LIN {X 0,Y 520.9,Z 965.477,A -85,B 0,C 180,E1 12388.23,E2 12388.23} C_VEL
LIN {X 0,Y 527.511,Z 989.341,A -85,B 0,C 180,E1 12389.551,E2 12389.551} C_VEL
LIN {X 0,Y 523.84,Z 1027.553,A -85,B 0,C 180,E1 12391.504,E2 12391.504} C_VEL
LIN {X 0,Y 519.786,Z 1062.879,A -85,B 0,C 180,E1 12394.029,E2 12394.029} C_VEL
LIN {X 0,Y 515.868,Z 1094.861,A -85,B 0,C 180,E1 12397.118,E2 12397.118} C_VEL
LIN {X 0,Y 512.363,Z 1122.894,A -85,B 0,C 180,E1 12400.744,E2 12400.744} C_VEL
LIN {X 0,Y 509.855,Z 1145.557,A -85,B 0,C 180,E1 12404.748,E2 12404.748} C_VEL
LIN {X 0,Y 508.379,Z 1161.603,A -85,B 0,C 180,E1 12408.676,E2 12408.676} C_VEL
LIN {X 0,Y 507.524,Z 1173.609,A -85,B 0,C 180,E1 12413.158,E2 12413.158} C_VEL
LIN {X 0,Y 507.269,Z 1178.777,A -85,B 0,C 180,E1 12416.583,E2 12416.583} C_VEL
LIN {X 0,Y 507.149,Z 1180.724,A -85,B 0,C 180,E1 12419.998,E2 12419.998} C_VEL
LIN {X 0,Y 507.304,Z 1179.309,A -85,B 0,C 180,E1 12423.414,E2 12423.414} C_VEL
LIN {X 0,Y 507.847,Z 1172.983,A -85,B 0,C 180,E1 12427.693,E2 12427.693} C_VEL
LIN {X 0,Y 508.836,Z 1161.151,A -85,B 0,C 180,E1 12431.996,E2 12431.996} C_VEL
LIN {X 0,Y 510.794,Z 1143.685,A -85,B 0,C 180,E1 12436.18,E2 12436.18} C_VEL
LIN {X 0,Y 513.724,Z 1121.065,A -85,B 0,C 180,E1 12440.059,E2 12440.059} C_VEL
LIN {X 0,Y 517.458,Z 1094.082,A -85,B 0,C 180,E1 12443.494,E2 12443.494} C_VEL
LIN {X 0,Y 521.913,Z 1061.989,A -85,B 0,C 180,E1 12446.546,E2 12446.546} C_VEL
LIN {X 0,Y 526.403,Z 1024.953,A -85,B 0,C 180,E1 12449.129,E2 12449.129} C_VEL
LIN {X 0,Y 529.643,Z 987.235,A -85,B 0,C 180,E1 12451.052,E2 12451.052} C_VEL
LIN {X 0,Y 522.519,Z 958.525,A -85,B 0,C 180,E1 12452.917,E2 12452.917} C_VEL
LIN {X 0,Y 511.608,Z 934.411,A -85,B 0,C 180,E1 12454.931,E2 12454.931} C_VEL
LIN {X 0,Y 505.831,Z 924.14,A -85,B 0,C 180,E1 12456.044,E2 12456.044} C_VEL
LIN {X 0,Y 505.742,Z 923.03,A -85,B 0,C 180,E1 12456.255,E2 12456.255} C_VEL
LIN {X 0,Y 505.562,Z 923.03,A -85,B 0,C 180,E1 12461.677,E2 12461.677} C_VEL
LIN {X 0,Y 505.58,Z 923.03,A -85,B 0,C 180,E1 12468.346,E2 12468.346} C_VEL
LIN {X 0,Y 505.778,Z 923.5,A -85,B 0,C 180,E1 12473,E2 12473} C_VEL
LIN {X 0,Y 508.487,Z 928.998,A -85,B 0,C 180,E1 12473.585,E2 12473.585} C_VEL
LIN {X 0,Y 520.191,Z 951.391,A -85,B 0,C 180,E1 12475.641,E2 12475.641} C_VEL
LIN {X 0,Y 529.457,Z 976.982,A -85,B 0,C 180,E1 12477.182,E2 12477.182} C_VEL
LIN {X 0,Y 531.635,Z 989.961,A -85,B 0,C 180,E1 12477.756,E2 12477.756} C_VEL
LIN {X 0,Y 527.643,Z 1032.457,A -85,B 0,C 180,E1 12479.219,E2 12479.219} C_VEL
LIN {X 0,Y 523.137,Z 1072.758,A -85,B 0,C 180,E1 12481.282,E2 12481.282} C_VEL
LIN {X 0,Y 518.67,Z 1110.607,A -85,B 0,C 180,E1 12483.99,E2 12483.99} C_VEL
LIN {X 0,Y 514.873,Z 1141.401,A -85,B 0,C 180,E1 12486.934,E2 12486.934} C_VEL
LIN {X 0,Y 509.62,Z 1153.637,A -85,B 0,C 180,E1 12488.212,E2 12488.212} C_VEL
LIN {X 0,Y 504.32,Z 1165.107,A -85,B 0,C 180,E1 12489.59,E2 12489.59} C_VEL
LIN {X 0,Y 501.753,Z 1188.474,A -85,B 0,C 180,E1 12493.393,E2 12493.393} C_VEL
LIN {X 0,Y 500.297,Z 1206.459,A -85,B 0,C 180,E1 12497.368,E2 12497.368} C_VEL
LIN {X 0,Y 499.642,Z 1218.968,A -85,B 0,C 180,E1 12501.319,E2 12501.319} C_VEL
LIN {X 0,Y 499.431,Z 1227.195,A -85,B 0,C 180,E1 12505.678,E2 12505.678} C_VEL
LIN {X 0,Y 499.394,Z 1229.924,A -85,B 0,C 180,E1 12510.015,E2 12510.015} C_VEL
LIN {X 0,Y 499.406,Z 1227.246,A -85,B 0,C 180,E1 12514.353,E2 12514.353} C_VEL
LIN {X 0,Y 499.659,Z 1219.037,A -85,B 0,C 180,E1 12518.712,E2 12518.712} C_VEL
LIN {X 0,Y 500.448,Z 1204.807,A -85,B 0,C 180,E1 12523.103,E2 12523.103} C_VEL
LIN {X 0,Y 502.2,Z 1184.844,A -85,B 0,C 180,E1 12527.3,E2 12527.3} C_VEL
LIN {X 0,Y 504.951,Z 1160.393,A -85,B 0,C 180,E1 12531.059,E2 12531.059} C_VEL
LIN {X 0,Y 508.606,Z 1130.776,A -85,B 0,C 180,E1 12534.476,E2 12534.476} C_VEL
LIN {X 0,Y 512.785,Z 1097.991,A -85,B 0,C 180,E1 12537.311,E2 12537.311} C_VEL
LIN {X 0,Y 517.104,Z 1059.799,A -85,B 0,C 180,E1 12539.735,E2 12539.735} C_VEL
LIN {X 0,Y 520.912,Z 1019.258,A -85,B 0,C 180,E1 12541.491,E2 12541.491} C_VEL
LIN {X 0,Y 522.653,Z 988.371,A -85,B 0,C 180,E1 12542.388,E2 12542.388} C_VEL
LIN {X 0,Y 497.906,Z 923.03,A -85,B 0,C 180,E1 12545.137,E2 12545.137} C_VEL
LIN {X 0,Y 497.67,Z 923.03,A -85,B 0,C 180,E1 12551.928,E2 12551.928} C_VEL
LIN {X 0,Y 497.676,Z 923.03,A -85,B 0,C 180,E1 12558.091,E2 12558.091} C_VEL
LIN {X 0,Y 497.784,Z 923.03,A -85,B 0,C 180,E1 12564.778,E2 12564.778} C_VEL
LIN {X 0,Y 497.927,Z 923.03,A -85,B 0,C 180,E1 12570.953,E2 12570.953} C_VEL
LIN {X 0,Y 498.06,Z 923.03,A -85,B 0,C 180,E1 12576.773,E2 12576.773} C_VEL
LIN {X 0,Y 498.161,Z 923.03,A -85,B 0,C 180,E1 12582.344,E2 12582.344} C_VEL
LIN {X 0,Y 498.445,Z 923.03,A -85,B 0,C 180,E1 12587.75,E2 12587.75} C_VEL
LIN {X 0,Y 498.675,Z 923.03,A -85,B 0,C 180,E1 12590.677,E2 12590.677} C_VEL
LIN {X 0,Y 508.907,Z 958.608,A -85,B 0,C 180,E1 12591.929,E2 12591.929} C_VEL
LIN {X 0,Y 508.728,Z 999.028,A -85,B 0,C 180,E1 12592.833,E2 12592.833} C_VEL
LIN {X 0,Y 507.812,Z 1027.625,A -85,B 0,C 180,E1 12594.131,E2 12594.131} C_VEL
LIN {X 0,Y 506.287,Z 1053.415,A -85,B 0,C 180,E1 12596.044,E2 12596.044} C_VEL
LIN {X 0,Y 504.623,Z 1075.233,A -85,B 0,C 180,E1 12598.5,E2 12598.5} C_VEL
LIN {X 0,Y 503.071,Z 1091.622,A -85,B 0,C 180,E1 12601.293,E2 12601.293} C_VEL
LIN {X 0,Y 501.81,Z 1102.595,A -85,B 0,C 180,E1 12604.319,E2 12604.319} C_VEL
LIN {X 0,Y 501.149,Z 1107.533,A -85,B 0,C 180,E1 12606.929,E2 12606.929} C_VEL
LIN {X 0,Y 500.871,Z 1108.785,A -85,B 0,C 180,E1 12608.678,E2 12608.678} C_VEL
LIN {X 0,Y 500.809,Z 1107.29,A -85,B 0,C 180,E1 12611.485,E2 12611.485} C_VEL
LIN {X 0,Y 501.096,Z 1100.753,A -85,B 0,C 180,E1 12614.58,E2 12614.58} C_VEL
LIN {X 0,Y 501.602,Z 1089.12,A -85,B 0,C 180,E1 12617.535,E2 12617.535} C_VEL
LIN {X 0,Y 502.57,Z 1070.875,A -85,B 0,C 180,E1 12620.461,E2 12620.461} C_VEL
LIN {X 0,Y 503.728,Z 1048.712,A -85,B 0,C 180,E1 12622.843,E2 12622.843} C_VEL
LIN {X 0,Y 504.947,Z 1021.724,A -85,B 0,C 180,E1 12624.771,E2 12624.771} C_VEL
LIN {X 0,Y 505.662,Z 992.567,A -85,B 0,C 180,E1 12626.047,E2 12626.047} C_VEL
LIN {X 0,Y 505.274,Z 955.718,A -85,B 0,C 180,E1 12626.834,E2 12626.834} C_VEL
LIN {X 0,Y 498.179,Z 923.03,A -85,B 0,C 180,E1 12627.573,E2 12627.573} C_VEL
LIN {X 0,Y 497.791,Z 923.03,A -85,B 0,C 180,E1 12633.123,E2 12633.123} C_VEL
LIN {X 0,Y 497.681,Z 923.03,A -85,B 0,C 180,E1 12639.617,E2 12639.617} C_VEL
LIN {X 0,Y 497.669,Z 923.03,A -85,B 0,C 180,E1 12645.688,E2 12645.688} C_VEL
LIN {X 0,Y 497.713,Z 923.03,A -85,B 0,C 180,E1 12652.131,E2 12652.131} C_VEL
LIN {X 0,Y 497.801,Z 923.03,A -85,B 0,C 180,E1 12658.21,E2 12658.21} C_VEL
LIN {X 0,Y 498.065,Z 923.03,A -85,B 0,C 180,E1 12662.915,E2 12662.915} C_VEL
LIN {X 0,Y 498.194,Z 923.03,A -85,B 0,C 180,E1 12668.641,E2 12668.641} C_VEL
LIN {X 0,Y 498.358,Z 923.03,A -85,B 0,C 180,E1 12674.149,E2 12674.149} C_VEL
LIN {X 0,Y 498.609,Z 923.03,A -85,B 0,C 180,E1 12679.509,E2 12679.509} C_VEL
LIN {X 0,Y 498.918,Z 923.03,A -85,B 0,C 180,E1 12684.772,E2 12684.772} C_VEL
LIN {X 0,Y 499.243,Z 923.03,A -85,B 0,C 180,E1 12689.985,E2 12689.985} C_VEL
LIN {X 0,Y 498.995,Z 923.03,A -85,B 0,C 180,E1 12695.197,E2 12695.197} C_VEL
LIN {X 0,Y 498.647,Z 923.03,A -85,B 0,C 180,E1 12700.459,E2 12700.459} C_VEL
LIN {X 0,Y 498.446,Z 923.03,A -85,B 0,C 180,E1 12705.816,E2 12705.816} C_VEL
LIN {X 0,Y 498.223,Z 923.03,A -85,B 0,C 180,E1 12711.325,E2 12711.325} C_VEL
LIN {X 0,Y 498.034,Z 923.03,A -85,B 0,C 180,E1 12717.053,E2 12717.053} C_VEL
LIN {X 0,Y 497.906,Z 923.03,A -85,B 0,C 180,E1 12723.091,E2 12723.091} C_VEL
LIN {X 0,Y 497.714,Z 923.03,A -85,B 0,C 180,E1 12729.587,E2 12729.587} C_VEL
LIN {X 0,Y 497.783,Z 923.03,A -85,B 0,C 180,E1 12735.715,E2 12735.715} C_VEL
LIN {X 0,Y 497.69,Z 923.03,A -85,B 0,C 180,E1 12742.099,E2 12742.099} C_VEL
LIN {X 0,Y 497.85,Z 923.03,A -85,B 0,C 180,E1 12745.723,E2 12745.723} C_VEL
LIN {X 0,Y 513.789,Z 967.903,A -85,B 0,C 180,E1 12747.939,E2 12747.939} C_VEL
LIN {X 0,Y 520.205,Z 990.832,A -85,B 0,C 180,E1 12749.252,E2 12749.252} C_VEL
LIN {X 0,Y 516.455,Z 1028.551,A -85,B 0,C 180,E1 12751.22,E2 12751.22} C_VEL
LIN {X 0,Y 512.346,Z 1063.303,A -85,B 0,C 180,E1 12753.741,E2 12753.741} C_VEL
LIN {X 0,Y 508.279,Z 1095.425,A -85,B 0,C 180,E1 12756.888,E2 12756.888} C_VEL
LIN {X 0,Y 504.693,Z 1123.137,A -85,B 0,C 180,E1 12760.521,E2 12760.521} C_VEL
LIN {X 0,Y 502.177,Z 1145.041,A -85,B 0,C 180,E1 12764.401,E2 12764.401} C_VEL
LIN {X 0,Y 500.557,Z 1161.737,A -85,B 0,C 180,E1 12768.497,E2 12768.497} C_VEL
LIN {X 0,Y 499.648,Z 1173.871,A -85,B 0,C 180,E1 12773.05,E2 12773.05} C_VEL
LIN {X 0,Y 499.399,Z 1179.11,A -85,B 0,C 180,E1 12776.529,E2 12776.529} C_VEL
LIN {X 0,Y 499.26,Z 1181.117,A -85,B 0,C 180,E1 12779.998,E2 12779.998} C_VEL
LIN {X 0,Y 499.443,Z 1179.682,A -85,B 0,C 180,E1 12783.555,E2 12783.555} C_VEL
LIN {X 0,Y 500.017,Z 1173.488,A -85,B 0,C 180,E1 12787.814,E2 12787.814} C_VEL
LIN {X 0,Y 501.069,Z 1161.701,A -85,B 0,C 180,E1 12792.185,E2 12792.185} C_VEL
LIN {X 0,Y 503.14,Z 1144.341,A -85,B 0,C 180,E1 12796.421,E2 12796.421} C_VEL
LIN {X 0,Y 506.144,Z 1122.627,A -85,B 0,C 180,E1 12800.233,E2 12800.233} C_VEL
LIN {X 0,Y 510.032,Z 1096.118,A -85,B 0,C 180,E1 12803.704,E2 12803.704} C_VEL
LIN {X 0,Y 514.733,Z 1064.179,A -85,B 0,C 180,E1 12806.829,E2 12806.829} C_VEL
LIN {X 0,Y 519.594,Z 1026.686,A -85,B 0,C 180,E1 12809.524,E2 12809.524} C_VEL
LIN {X 0,Y 523.222,Z 990.214,A -85,B 0,C 180,E1 12811.431,E2 12811.431} C_VEL
LIN {X 0,Y 516.536,Z 961.811,A -85,B 0,C 180,E1 12813.365,E2 12813.365} C_VEL
LIN {X 0,Y 506.625,Z 939.472,A -85,B 0,C 180,E1 12815.366,E2 12815.366} C_VEL
LIN {X 0,Y 499.796,Z 928.28,A -85,B 0,C 180,E1 12816.779,E2 12816.779} C_VEL
LIN {X 0,Y 497.709,Z 923.03,A -85,B 0,C 180,E1 12817.386,E2 12817.386} C_VEL
LIN {X 0,Y 497.639,Z 923.03,A -85,B 0,C 180,E1 12823.245,E2 12823.245} C_VEL
LIN {X 0,Y 497.675,Z 923.03,A -85,B 0,C 180,E1 12829.38,E2 12829.38} C_VEL
LIN {X 0,Y 497.831,Z 923.176,A -85,B 0,C 180,E1 12831.72,E2 12831.72} C_VEL
LIN {X 0,Y 500.458,Z 928.905,A -85,B 0,C 180,E1 12832.418,E2 12832.418} C_VEL
LIN {X 0,Y 510.633,Z 946.873,A -85,B 0,C 180,E1 12834.465,E2 12834.465} C_VEL
LIN {X 0,Y 520.697,Z 970.847,A -85,B 0,C 180,E1 12836.241,E2 12836.241} C_VEL
LIN {X 0,Y 525.193,Z 990.447,A -85,B 0,C 180,E1 12837.265,E2 12837.265} C_VEL
LIN {X 0,Y 520.871,Z 1033.253,A -85,B 0,C 180,E1 12838.786,E2 12838.786} C_VEL
LIN {X 0,Y 516.081,Z 1073.316,A -85,B 0,C 180,E1 12840.891,E2 12840.891} C_VEL
LIN {X 0,Y 511.285,Z 1111.61,A -85,B 0,C 180,E1 12843.703,E2 12843.703} C_VEL
LIN {X 0,Y 506.983,Z 1144.642,A -85,B 0,C 180,E1 12846.989,E2 12846.989} C_VEL
LIN {X 0,Y 504.32,Z 1165.107,A -85,B 0,C 180,E1 12849.59,E2 12849.59} C_VEL
LIN {X 0,Y 499.297,Z 1175.816,A -85,B 0,C 180,E1 12851.071,E2 12851.071} C_VEL
LIN {X 0,Y 494.335,Z 1185.609,A -85,B 0,C 180,E1 12852.653,E2 12852.653} C_VEL
LIN {X 0,Y 492.598,Z 1204.397,A -85,B 0,C 180,E1 12856.716,E2 12856.716} C_VEL
LIN {X 0,Y 491.748,Z 1218.588,A -85,B 0,C 180,E1 12861.178,E2 12861.178} C_VEL
LIN {X 0,Y 491.532,Z 1226.811,A -85,B 0,C 180,E1 12865.608,E2 12865.608} C_VEL
LIN {X 0,Y 491.519,Z 1229.511,A -85,B 0,C 180,E1 12870.016,E2 12870.016} C_VEL
LIN {X 0,Y 491.514,Z 1226.773,A -85,B 0,C 180,E1 12874.423,E2 12874.423} C_VEL
LIN {X 0,Y 491.768,Z 1218.467,A -85,B 0,C 180,E1 12878.853,E2 12878.853} C_VEL
LIN {X 0,Y 492.604,Z 1204.095,A -85,B 0,C 180,E1 12883.316,E2 12883.316} C_VEL
LIN {X 0,Y 494.46,Z 1183.965,A -85,B 0,C 180,E1 12887.579,E2 12887.579} C_VEL
LIN {X 0,Y 497.354,Z 1159.298,A -85,B 0,C 180,E1 12891.397,E2 12891.397} C_VEL
LIN {X 0,Y 501.179,Z 1129.375,A -85,B 0,C 180,E1 12894.863,E2 12894.863} C_VEL
LIN {X 0,Y 505.628,Z 1095.022,A -85,B 0,C 180,E1 12897.829,E2 12897.829} C_VEL
LIN {X 0,Y 510.132,Z 1056.206,A -85,B 0,C 180,E1 12900.251,E2 12900.251} C_VEL
LIN {X 0,Y 513.969,Z 1015.807,A -85,B 0,C 180,E1 12901.966,E2 12901.966} C_VEL
LIN {X 0,Y 515.199,Z 989.635,A -85,B 0,C 180,E1 12902.747,E2 12902.747} C_VEL
LIN {X 0,Y 489.896,Z 923.03,A -85,B 0,C 180,E1 12905.649,E2 12905.649} C_VEL
LIN {X 0,Y 489.777,Z 923.03,A -85,B 0,C 180,E1 12912.232,E2 12912.232} C_VEL
LIN {X 0,Y 489.782,Z 923.03,A -85,B 0,C 180,E1 12917.788,E2 12917.788} C_VEL
LIN {X 0,Y 489.789,Z 923.03,A -85,B 0,C 180,E1 12924.115,E2 12924.115} C_VEL
LIN {X 0,Y 489.939,Z 923.03,A -85,B 0,C 180,E1 12930.433,E2 12930.433} C_VEL
LIN {X 0,Y 490.138,Z 923.03,A -85,B 0,C 180,E1 12936.374,E2 12936.374} C_VEL
LIN {X 0,Y 490.226,Z 923.03,A -85,B 0,C 180,E1 12942.049,E2 12942.049} C_VEL
LIN {X 0,Y 490.529,Z 923.03,A -85,B 0,C 180,E1 12947.549,E2 12947.549} C_VEL
LIN {X 0,Y 490.761,Z 923.03,A -85,B 0,C 180,E1 12950.227,E2 12950.227} C_VEL
LIN {X 0,Y 501.478,Z 958.867,A -85,B 0,C 180,E1 12951.563,E2 12951.563} C_VEL
LIN {X 0,Y 501.419,Z 1000.68,A -85,B 0,C 180,E1 12952.537,E2 12952.537} C_VEL
LIN {X 0,Y 500.35,Z 1030.37,A -85,B 0,C 180,E1 12953.934,E2 12953.934} C_VEL
LIN {X 0,Y 498.768,Z 1055.583,A -85,B 0,C 180,E1 12955.876,E2 12955.876} C_VEL
LIN {X 0,Y 497.05,Z 1076.203,A -85,B 0,C 180,E1 12958.26,E2 12958.26} C_VEL
LIN {X 0,Y 495.413,Z 1092.633,A -85,B 0,C 180,E1 12961.094,E2 12961.094} C_VEL
LIN {X 0,Y 494.157,Z 1103.017,A -85,B 0,C 180,E1 12963.947,E2 12963.947} C_VEL
LIN {X 0,Y 493.3,Z 1108.793,A -85,B 0,C 180,E1 12967.04,E2 12967.04} C_VEL
LIN {X 0,Y 493.026,Z 1109.785,A -85,B 0,C 180,E1 12968.817,E2 12968.817} C_VEL
LIN {X 0,Y 492.963,Z 1108.591,A -85,B 0,C 180,E1 12971.162,E2 12971.162} C_VEL
LIN {X 0,Y 493.281,Z 1101.236,A -85,B 0,C 180,E1 12974.736,E2 12974.736} C_VEL
LIN {X 0,Y 493.84,Z 1088.774,A -85,B 0,C 180,E1 12977.82,E2 12977.82} C_VEL
LIN {X 0,Y 494.756,Z 1071.6,A -85,B 0,C 180,E1 12980.565,E2 12980.565} C_VEL
LIN {X 0,Y 495.946,Z 1049.345,A -85,B 0,C 180,E1 12982.98,E2 12982.98} C_VEL
LIN {X 0,Y 497.22,Z 1022.145,A -85,B 0,C 180,E1 12984.941,E2 12984.941} C_VEL
LIN {X 0,Y 497.97,Z 992.413,A -85,B 0,C 180,E1 12986.242,E2 12986.242} C_VEL
LIN {X 0,Y 497.517,Z 956.432,A -85,B 0,C 180,E1 12987.02,E2 12987.02} C_VEL
LIN {X 0,Y 490.261,Z 923.03,A -85,B 0,C 180,E1 12987.835,E2 12987.835} C_VEL
LIN {X 0,Y 489.841,Z 923.03,A -85,B 0,C 180,E1 12993.732,E2 12993.732} C_VEL
LIN {X 0,Y 489.744,Z 923.03,A -85,B 0,C 180,E1 13000.39,E2 13000.39} C_VEL
LIN {X 0,Y 489.748,Z 923.03,A -85,B 0,C 180,E1 13005.21,E2 13005.21} C_VEL
LIN {X 0,Y 489.79,Z 923.03,A -85,B 0,C 180,E1 13010.474,E2 13010.474} C_VEL
LIN {X 0,Y 489.866,Z 923.03,A -85,B 0,C 180,E1 13016.398,E2 13016.398} C_VEL
LIN {X 0,Y 490.14,Z 923.03,A -85,B 0,C 180,E1 13022.44,E2 13022.44} C_VEL
LIN {X 0,Y 490.238,Z 923.03,A -85,B 0,C 180,E1 13028.277,E2 13028.277} C_VEL
LIN {X 0,Y 490.425,Z 923.03,A -85,B 0,C 180,E1 13033.886,E2 13033.886} C_VEL
LIN {X 0,Y 490.703,Z 923.03,A -85,B 0,C 180,E1 13040.217,E2 13040.217} C_VEL
LIN {X 0,Y 491.184,Z 923.03,A -85,B 0,C 180,E1 13046.457,E2 13046.457} C_VEL
LIN {X 0,Y 491.242,Z 923.03,A -85,B 0,C 180,E1 13051.747,E2 13051.747} C_VEL
LIN {X 0,Y 490.928,Z 923.03,A -85,B 0,C 180,E1 13057.056,E2 13057.056} C_VEL
LIN {X 0,Y 490.638,Z 923.03,A -85,B 0,C 180,E1 13062.433,E2 13062.433} C_VEL
LIN {X 0,Y 490.452,Z 923.03,A -85,B 0,C 180,E1 13067.927,E2 13067.927} C_VEL
LIN {X 0,Y 490.187,Z 923.03,A -85,B 0,C 180,E1 13073.606,E2 13073.606} C_VEL
LIN {X 0,Y 490.035,Z 923.03,A -85,B 0,C 180,E1 13079.542,E2 13079.542} C_VEL
LIN {X 0,Y 489.849,Z 923.03,A -85,B 0,C 180,E1 13085.859,E2 13085.859} C_VEL
LIN {X 0,Y 489.843,Z 923.03,A -85,B 0,C 180,E1 13092.235,E2 13092.235} C_VEL
LIN {X 0,Y 489.826,Z 923.03,A -85,B 0,C 180,E1 13097.736,E2 13097.736} C_VEL
LIN {X 0,Y 489.802,Z 923.03,A -85,B 0,C 180,E1 13104.112,E2 13104.112} C_VEL
LIN {X 0,Y 489.953,Z 923.03,A -85,B 0,C 180,E1 13105.27,E2 13105.27} C_VEL
LIN {X 0,Y 505.455,Z 966.663,A -85,B 0,C 180,E1 13107.442,E2 13107.442} C_VEL
LIN {X 0,Y 512.877,Z 992.665,A -85,B 0,C 180,E1 13108.964,E2 13108.964} C_VEL
LIN {X 0,Y 508.997,Z 1030.048,A -85,B 0,C 180,E1 13110.964,E2 13110.964} C_VEL
LIN {X 0,Y 504.736,Z 1064.796,A -85,B 0,C 180,E1 13113.542,E2 13113.542} C_VEL
LIN {X 0,Y 500.661,Z 1096.044,A -85,B 0,C 180,E1 13116.661,E2 13116.661} C_VEL
LIN {X 0,Y 496.895,Z 1124.411,A -85,B 0,C 180,E1 13120.455,E2 13120.455} C_VEL
LIN {X 0,Y 494.239,Z 1146.618,A -85,B 0,C 180,E1 13124.51,E2 13124.51} C_VEL
LIN {X 0,Y 492.592,Z 1163.68,A -85,B 0,C 180,E1 13128.898,E2 13128.898} C_VEL
LIN {X 0,Y 491.755,Z 1174.346,A -85,B 0,C 180,E1 13133.059,E2 13133.059} C_VEL
LIN {X 0,Y 491.509,Z 1179.44,A -85,B 0,C 180,E1 13136.473,E2 13136.473} C_VEL
LIN {X 0,Y 491.384,Z 1181.51,A -85,B 0,C 180,E1 13139.998,E2 13139.998} C_VEL
LIN {X 0,Y 491.573,Z 1180.229,A -85,B 0,C 180,E1 13143.523,E2 13143.523} C_VEL
LIN {X 0,Y 492.192,Z 1174.01,A -85,B 0,C 180,E1 13147.939,E2 13147.939} C_VEL
LIN {X 0,Y 493.305,Z 1162.282,A -85,B 0,C 180,E1 13152.38,E2 13152.38} C_VEL
LIN {X 0,Y 495.439,Z 1145.611,A -85,B 0,C 180,E1 13156.553,E2 13156.553} C_VEL
LIN {X 0,Y 498.647,Z 1123.707,A -85,B 0,C 180,E1 13160.495,E2 13160.495} C_VEL
LIN {X 0,Y 502.77,Z 1097.339,A -85,B 0,C 180,E1 13164.023,E2 13164.023} C_VEL
LIN {X 0,Y 507.56,Z 1066.513,A -85,B 0,C 180,E1 13167.12,E2 13167.12} C_VEL
LIN {X 0,Y 512.611,Z 1030.588,A -85,B 0,C 180,E1 13169.803,E2 13169.803} C_VEL
LIN {X 0,Y 516.8,Z 992.75,A -85,B 0,C 180,E1 13171.86,E2 13171.86} C_VEL
LIN {X 0,Y 510.765,Z 965.636,A -85,B 0,C 180,E1 13173.801,E2 13173.801} C_VEL
LIN {X 0,Y 501.844,Z 944.59,A -85,B 0,C 180,E1 13175.8,E2 13175.8} C_VEL
LIN {X 0,Y 493.231,Z 929.547,A -85,B 0,C 180,E1 13177.858,E2 13177.858} C_VEL
LIN {X 0,Y 489.818,Z 924.221,A -85,B 0,C 180,E1 13178.864,E2 13178.864} C_VEL
LIN {X 0,Y 489.708,Z 923.03,A -85,B 0,C 180,E1 13179.07,E2 13179.07} C_VEL
LIN {X 0,Y 489.717,Z 923.03,A -85,B 0,C 180,E1 13185.208,E2 13185.208} C_VEL
LIN {X 0,Y 489.802,Z 923.705,A -85,B 0,C 180,E1 13190.129,E2 13190.129} C_VEL
LIN {X 0,Y 492.66,Z 929.066,A -85,B 0,C 180,E1 13191.053,E2 13191.053} C_VEL
LIN {X 0,Y 498.519,Z 938.706,A -85,B 0,C 180,E1 13192.532,E2 13192.532} C_VEL
LIN {X 0,Y 507.556,Z 955.699,A -85,B 0,C 180,E1 13194.388,E2 13194.388} C_VEL
LIN {X 0,Y 516.046,Z 978.486,A -85,B 0,C 180,E1 13196.046,E2 13196.046} C_VEL
LIN {X 0,Y 518.717,Z 992.734,A -85,B 0,C 180,E1 13196.804,E2 13196.804} C_VEL
LIN {X 0,Y 514.061,Z 1035.231,A -85,B 0,C 180,E1 13198.385,E2 13198.385} C_VEL
LIN {X 0,Y 508.725,Z 1076.892,A -85,B 0,C 180,E1 13200.672,E2 13200.672} C_VEL
LIN {X 0,Y 503.789,Z 1113.324,A -85,B 0,C 180,E1 13203.468,E2 13203.468} C_VEL
LIN {X 0,Y 499.546,Z 1144.327,A -85,B 0,C 180,E1 13206.627,E2 13206.627} C_VEL
LIN {X 0,Y 496.093,Z 1171.092,A -85,B 0,C 180,E1 13210.21,E2 13210.21} C_VEL
LIN {X 0,Y 494.335,Z 1185.609,A -85,B 0,C 180,E1 13212.653,E2 13212.653} C_VEL
LIN {X 0,Y 489.503,Z 1194.505,A -85,B 0,C 180,E1 13214.325,E2 13214.325} C_VEL
LIN {X 0,Y 484.896,Z 1202.458,A -85,B 0,C 180,E1 13216.086,E2 13216.086} C_VEL
LIN {X 0,Y 483.913,Z 1217.235,A -85,B 0,C 180,E1 13220.62,E2 13220.62} C_VEL
LIN {X 0,Y 483.664,Z 1225.235,A -85,B 0,C 180,E1 13224.638,E2 13224.638} C_VEL
LIN {X 0,Y 483.6,Z 1228.726,A -85,B 0,C 180,E1 13228.225,E2 13228.225} C_VEL
LIN {X 0,Y 483.682,Z 1228.608,A -85,B 0,C 180,E1 13231.806,E2 13231.806} C_VEL
LIN {X 0,Y 483.72,Z 1223.59,A -85,B 0,C 180,E1 13236.292,E2 13236.292} C_VEL
LIN {X 0,Y 484.119,Z 1212.825,A -85,B 0,C 180,E1 13240.809,E2 13240.809} C_VEL
LIN {X 0,Y 485.244,Z 1198.121,A -85,B 0,C 180,E1 13244.809,E2 13244.809} C_VEL
LIN {X 0,Y 487.39,Z 1177.197,A -85,B 0,C 180,E1 13248.89,E2 13248.89} C_VEL
LIN {X 0,Y 490.708,Z 1151.297,A -85,B 0,C 180,E1 13252.633,E2 13252.633} C_VEL
LIN {X 0,Y 494.623,Z 1121.907,A -85,B 0,C 180,E1 13255.848,E2 13255.848} C_VEL
LIN {X 0,Y 498.992,Z 1088.763,A -85,B 0,C 180,E1 13258.577,E2 13258.577} C_VEL
LIN {X 0,Y 503.306,Z 1051.604,A -85,B 0,C 180,E1 13260.821,E2 13260.821} C_VEL
LIN {X 0,Y 507.125,Z 1010.92,A -85,B 0,C 180,E1 13262.499,E2 13262.499} C_VEL
LIN {X 0,Y 508.143,Z 992.06,A -85,B 0,C 180,E1 13263.057,E2 13263.057} C_VEL
LIN {X 0,Y 483.211,Z 927.294,A -85,B 0,C 180,E1 13265.922,E2 13265.922} C_VEL
LIN {X 0,Y 481.949,Z 923.03,A -85,B 0,C 180,E1 13266.12,E2 13266.12} C_VEL
LIN {X 0,Y 481.8,Z 923.03,A -85,B 0,C 180,E1 13271.212,E2 13271.212} C_VEL
LIN {X 0,Y 481.787,Z 923.03,A -85,B 0,C 180,E1 13276.371,E2 13276.371} C_VEL
LIN {X 0,Y 481.886,Z 923.03,A -85,B 0,C 180,E1 13281.642,E2 13281.642} C_VEL
LIN {X 0,Y 481.95,Z 923.03,A -85,B 0,C 180,E1 13287.86,E2 13287.86} C_VEL
LIN {X 0,Y 482.183,Z 923.03,A -85,B 0,C 180,E1 13293.979,E2 13293.979} C_VEL
LIN {X 0,Y 482.334,Z 923.03,A -85,B 0,C 180,E1 13300.061,E2 13300.061} C_VEL
LIN {X 0,Y 482.498,Z 923.03,A -85,B 0,C 180,E1 13306.179,E2 13306.179} C_VEL
LIN {X 0,Y 482.812,Z 923.03,A -85,B 0,C 180,E1 13309.732,E2 13309.732} C_VEL
LIN {X 0,Y 494.016,Z 959.021,A -85,B 0,C 180,E1 13311.172,E2 13311.172} C_VEL
LIN {X 0,Y 494.18,Z 1000.314,A -85,B 0,C 180,E1 13312.148,E2 13312.148} C_VEL
LIN {X 0,Y 493.137,Z 1029.61,A -85,B 0,C 180,E1 13313.514,E2 13313.514} C_VEL
LIN {X 0,Y 491.416,Z 1055.459,A -85,B 0,C 180,E1 13315.483,E2 13315.483} C_VEL
LIN {X 0,Y 489.536,Z 1077.264,A -85,B 0,C 180,E1 13318.012,E2 13318.012} C_VEL
LIN {X 0,Y 487.759,Z 1093.645,A -85,B 0,C 180,E1 13320.889,E2 13320.889} C_VEL
LIN {X 0,Y 486.336,Z 1104.642,A -85,B 0,C 180,E1 13324.011,E2 13324.011} C_VEL
LIN {X 0,Y 485.463,Z 1110.003,A -85,B 0,C 180,E1 13327.154,E2 13327.154} C_VEL
LIN {X 0,Y 485.198,Z 1110.763,A -85,B 0,C 180,E1 13328.96,E2 13328.96} C_VEL
LIN {X 0,Y 485.14,Z 1109.269,A -85,B 0,C 180,E1 13331.344,E2 13331.344} C_VEL
LIN {X 0,Y 485.435,Z 1101.959,A -85,B 0,C 180,E1 13334.805,E2 13334.805} C_VEL
LIN {X 0,Y 486.016,Z 1089.602,A -85,B 0,C 180,E1 13337.882,E2 13337.882} C_VEL
LIN {X 0,Y 487.018,Z 1071.782,A -85,B 0,C 180,E1 13340.746,E2 13340.746} C_VEL
LIN {X 0,Y 488.222,Z 1048.586,A -85,B 0,C 180,E1 13343.245,E2 13343.245} C_VEL
LIN {X 0,Y 489.497,Z 1021.788,A -85,B 0,C 180,E1 13345.161,E2 13345.161} C_VEL
LIN {X 0,Y 490.254,Z 991.188,A -85,B 0,C 180,E1 13346.48,E2 13346.48} C_VEL
LIN {X 0,Y 489.731,Z 957.005,A -85,B 0,C 180,E1 13347.21,E2 13347.21} C_VEL
LIN {X 0,Y 482.322,Z 923.03,A -85,B 0,C 180,E1 13348.033,E2 13348.033} C_VEL
LIN {X 0,Y 481.852,Z 923.03,A -85,B 0,C 180,E1 13354.369,E2 13354.369} C_VEL
LIN {X 0,Y 481.834,Z 923.03,A -85,B 0,C 180,E1 13358.848,E2 13358.848} C_VEL
LIN {X 0,Y 481.785,Z 923.03,A -85,B 0,C 180,E1 13363.814,E2 13363.814} C_VEL
LIN {X 0,Y 481.84,Z 923.03,A -85,B 0,C 180,E1 13368.825,E2 13368.825} C_VEL
LIN {X 0,Y 481.865,Z 923.03,A -85,B 0,C 180,E1 13374.625,E2 13374.625} C_VEL
LIN {X 0,Y 482.069,Z 923.03,A -85,B 0,C 180,E1 13379.883,E2 13379.883} C_VEL
LIN {X 0,Y 482.242,Z 923.03,A -85,B 0,C 180,E1 13385.946,E2 13385.946} C_VEL
LIN {X 0,Y 482.462,Z 923.03,A -85,B 0,C 180,E1 13391.733,E2 13391.733} C_VEL
LIN {X 0,Y 482.653,Z 923.03,A -85,B 0,C 180,E1 13397.326,E2 13397.326} C_VEL
LIN {X 0,Y 482.98,Z 923.03,A -85,B 0,C 180,E1 13402.795,E2 13402.795} C_VEL
LIN {X 0,Y 483.296,Z 923.03,A -85,B 0,C 180,E1 13408.193,E2 13408.193} C_VEL
LIN {X 0,Y 483.187,Z 923.03,A -85,B 0,C 180,E1 13413.57,E2 13413.57} C_VEL
LIN {X 0,Y 482.918,Z 923.03,A -85,B 0,C 180,E1 13418.984,E2 13418.984} C_VEL
LIN {X 0,Y 482.667,Z 923.03,A -85,B 0,C 180,E1 13424.487,E2 13424.487} C_VEL
LIN {X 0,Y 482.445,Z 923.03,A -85,B 0,C 180,E1 13430.135,E2 13430.135} C_VEL
LIN {X 0,Y 482.206,Z 923.03,A -85,B 0,C 180,E1 13436.002,E2 13436.002} C_VEL
LIN {X 0,Y 482.025,Z 923.03,A -85,B 0,C 180,E1 13442.182,E2 13442.182} C_VEL
LIN {X 0,Y 481.874,Z 923.03,A -85,B 0,C 180,E1 13448.817,E2 13448.817} C_VEL
LIN {X 0,Y 481.877,Z 923.03,A -85,B 0,C 180,E1 13453.84,E2 13453.84} C_VEL
LIN {X 0,Y 481.853,Z 923.03,A -85,B 0,C 180,E1 13458.807,E2 13458.807} C_VEL
LIN {X 0,Y 482.045,Z 923.632,A -85,B 0,C 180,E1 13464.82,E2 13464.82} C_VEL
LIN {X 0,Y 497.597,Z 966.695,A -85,B 0,C 180,E1 13467.006,E2 13467.006} C_VEL
LIN {X 0,Y 505.523,Z 994.406,A -85,B 0,C 180,E1 13468.668,E2 13468.668} C_VEL
LIN {X 0,Y 501.454,Z 1032.307,A -85,B 0,C 180,E1 13470.753,E2 13470.753} C_VEL
LIN {X 0,Y 496.989,Z 1067.864,A -85,B 0,C 180,E1 13473.478,E2 13473.478} C_VEL
LIN {X 0,Y 492.584,Z 1099.884,A -85,B 0,C 180,E1 13476.815,E2 13476.815} C_VEL
LIN {X 0,Y 488.956,Z 1126.333,A -85,B 0,C 180,E1 13480.505,E2 13480.505} C_VEL
LIN {X 0,Y 486.419,Z 1147.309,A -85,B 0,C 180,E1 13484.43,E2 13484.43} C_VEL
LIN {X 0,Y 484.752,Z 1163.784,A -85,B 0,C 180,E1 13488.716,E2 13488.716} C_VEL
LIN {X 0,Y 483.883,Z 1174.764,A -85,B 0,C 180,E1 13493.041,E2 13493.041} C_VEL
LIN {X 0,Y 483.625,Z 1179.766,A -85,B 0,C 180,E1 13496.415,E2 13496.415} C_VEL
LIN {X 0,Y 483.494,Z 1181.906,A -85,B 0,C 180,E1 13499.998,E2 13499.998} C_VEL
LIN {X 0,Y 483.695,Z 1180.702,A -85,B 0,C 180,E1 13503.58,E2 13503.58} C_VEL
LIN {X 0,Y 484.364,Z 1174.551,A -85,B 0,C 180,E1 13508.068,E2 13508.068} C_VEL
LIN {X 0,Y 485.548,Z 1162.895,A -85,B 0,C 180,E1 13512.581,E2 13512.581} C_VEL
LIN {X 0,Y 487.856,Z 1146.022,A -85,B 0,C 180,E1 13516.879,E2 13516.879} C_VEL
LIN {X 0,Y 491.386,Z 1123.696,A -85,B 0,C 180,E1 13520.944,E2 13520.944} C_VEL
LIN {X 0,Y 495.752,Z 1097.124,A -85,B 0,C 180,E1 13524.536,E2 13524.536} C_VEL
LIN {X 0,Y 501.065,Z 1065.274,A -85,B 0,C 180,E1 13527.744,E2 13527.744} C_VEL
LIN {X 0,Y 506.434,Z 1028.567,A -85,B 0,C 180,E1 13530.478,E2 13530.478} C_VEL
LIN {X 0,Y 510.302,Z 994.251,A -85,B 0,C 180,E1 13532.387,E2 13532.387} C_VEL
LIN {X 0,Y 504.958,Z 968.943,A -85,B 0,C 180,E1 13534.297,E2 13534.297} C_VEL
LIN {X 0,Y 496.056,Z 947.244,A -85,B 0,C 180,E1 13536.528,E2 13536.528} C_VEL
LIN {X 0,Y 488.764,Z 935.342,A -85,B 0,C 180,E1 13538.437,E2 13538.437} C_VEL
LIN {X 0,Y 485.202,Z 929.464,A -85,B 0,C 180,E1 13539.661,E2 13539.661} C_VEL
LIN {X 0,Y 481.838,Z 924.011,A -85,B 0,C 180,E1 13541.249,E2 13541.249} C_VEL
LIN {X 0,Y 481.835,Z 923.03,A -85,B 0,C 180,E1 13542.143,E2 13542.143} C_VEL
LIN {X 0,Y 481.889,Z 923.643,A -85,B 0,C 180,E1 13547.736,E2 13547.736} C_VEL
LIN {X 0,Y 484.763,Z 929.185,A -85,B 0,C 180,E1 13549.215,E2 13549.215} C_VEL
LIN {X 0,Y 486.695,Z 931.568,A -85,B 0,C 180,E1 13549.893,E2 13549.893} C_VEL
LIN {X 0,Y 493.596,Z 942.544,A -85,B 0,C 180,E1 13551.896,E2 13551.896} C_VEL
LIN {X 0,Y 503.006,Z 961.358,A -85,B 0,C 180,E1 13554.025,E2 13554.025} C_VEL
LIN {X 0,Y 510.766,Z 984.219,A -85,B 0,C 180,E1 13555.735,E2 13555.735} C_VEL
LIN {X 0,Y 512.286,Z 995.401,A -85,B 0,C 180,E1 13556.329,E2 13556.329} C_VEL
LIN {X 0,Y 506.957,Z 1039.705,A -85,B 0,C 180,E1 13558.076,E2 13558.076} C_VEL
LIN {X 0,Y 501.337,Z 1080.33,A -85,B 0,C 180,E1 13560.445,E2 13560.445} C_VEL
LIN {X 0,Y 496.171,Z 1116.328,A -85,B 0,C 180,E1 13563.336,E2 13563.336} C_VEL
LIN {X 0,Y 491.557,Z 1148.366,A -85,B 0,C 180,E1 13566.769,E2 13566.769} C_VEL
LIN {X 0,Y 487.705,Z 1176.682,A -85,B 0,C 180,E1 13570.837,E2 13570.837} C_VEL
LIN {X 0,Y 485.253,Z 1198.73,A -85,B 0,C 180,E1 13575.189,E2 13575.189} C_VEL
LIN {X 0,Y 484.896,Z 1202.458,A -85,B 0,C 180,E1 13576.086,E2 13576.086} C_VEL
LIN {X 0,Y 480.415,Z 1209.356,A -85,B 0,C 180,E1 13577.929,E2 13577.929} C_VEL
LIN {X 0,Y 476.126,Z 1215.22,A -85,B 0,C 180,E1 13579.846,E2 13579.846} C_VEL
LIN {X 0,Y 475.825,Z 1223.497,A -85,B 0,C 180,E1 13583.635,E2 13583.635} C_VEL
LIN {X 0,Y 475.705,Z 1228.324,A -85,B 0,C 180,E1 13588.196,E2 13588.196} C_VEL
LIN {X 0,Y 475.788,Z 1228.168,A -85,B 0,C 180,E1 13591.836,E2 13591.836} C_VEL
LIN {X 0,Y 475.832,Z 1223.061,A -85,B 0,C 180,E1 13596.397,E2 13596.397} C_VEL
LIN {X 0,Y 476.161,Z 1214.135,A -85,B 0,C 180,E1 13600.343,E2 13600.343} C_VEL
LIN {X 0,Y 477.292,Z 1198.938,A -85,B 0,C 180,E1 13604.687,E2 13604.687} C_VEL
LIN {X 0,Y 479.602,Z 1177.058,A -85,B 0,C 180,E1 13609.058,E2 13609.058} C_VEL
LIN {X 0,Y 483.119,Z 1150.259,A -85,B 0,C 180,E1 13612.974,E2 13612.974} C_VEL
LIN {X 0,Y 487.397,Z 1119.312,A -85,B 0,C 180,E1 13616.357,E2 13616.357} C_VEL
LIN {X 0,Y 492.156,Z 1084.011,A -85,B 0,C 180,E1 13619.225,E2 13619.225} C_VEL
LIN {X 0,Y 496.693,Z 1045.666,A -85,B 0,C 180,E1 13621.469,E2 13621.469} C_VEL
LIN {X 0,Y 500.496,Z 1004.846,A -85,B 0,C 180,E1 13623.063,E2 13623.063} C_VEL
LIN {X 0,Y 500.594,Z 992.73,A -85,B 0,C 180,E1 13623.447,E2 13623.447} C_VEL
LIN {X 0,Y 474.008,Z 923.03,A -85,B 0,C 180,E1 13626.697,E2 13626.697} C_VEL
LIN {X 0,Y 473.795,Z 923.03,A -85,B 0,C 180,E1 13632.818,E2 13632.818} C_VEL
LIN {X 0,Y 473.801,Z 923.03,A -85,B 0,C 180,E1 13637.954,E2 13637.954} C_VEL
LIN {X 0,Y 473.944,Z 923.03,A -85,B 0,C 180,E1 13642.872,E2 13642.872} C_VEL
LIN {X 0,Y 474.07,Z 923.03,A -85,B 0,C 180,E1 13649.409,E2 13649.409} C_VEL
LIN {X 0,Y 474.268,Z 923.03,A -85,B 0,C 180,E1 13655.533,E2 13655.533} C_VEL
LIN {X 0,Y 474.369,Z 923.03,A -85,B 0,C 180,E1 13661.427,E2 13661.427} C_VEL
LIN {X 0,Y 474.657,Z 923.03,A -85,B 0,C 180,E1 13667.126,E2 13667.126} C_VEL
LIN {X 0,Y 474.893,Z 923.061,A -85,B 0,C 180,E1 13669.226,E2 13669.226} C_VEL
LIN {X 0,Y 486.577,Z 959.368,A -85,B 0,C 180,E1 13670.764,E2 13670.764} C_VEL
LIN {X 0,Y 487.347,Z 976.227,A -85,B 0,C 180,E1 13671.157,E2 13671.157} C_VEL
LIN {X 0,Y 486.805,Z 1007.453,A -85,B 0,C 180,E1 13672.025,E2 13672.025} C_VEL
LIN {X 0,Y 485.615,Z 1034.298,A -85,B 0,C 180,E1 13673.413,E2 13673.413} C_VEL
LIN {X 0,Y 483.828,Z 1058.797,A -85,B 0,C 180,E1 13675.412,E2 13675.412} C_VEL
LIN {X 0,Y 481.859,Z 1079.876,A -85,B 0,C 180,E1 13677.98,E2 13677.98} C_VEL
LIN {X 0,Y 480.005,Z 1095.734,A -85,B 0,C 180,E1 13680.904,E2 13680.904} C_VEL
LIN {X 0,Y 478.69,Z 1105.073,A -85,B 0,C 180,E1 13683.622,E2 13683.622} C_VEL
LIN {X 0,Y 477.84,Z 1110.288,A -85,B 0,C 180,E1 13686.357,E2 13686.357} C_VEL
LIN {X 0,Y 477.352,Z 1111.743,A -85,B 0,C 180,E1 13689.109,E2 13689.109} C_VEL
LIN {X 0,Y 477.327,Z 1109.581,A -85,B 0,C 180,E1 13691.784,E2 13691.784} C_VEL
LIN {X 0,Y 477.614,Z 1102.07,A -85,B 0,C 180,E1 13695.054,E2 13695.054} C_VEL
LIN {X 0,Y 478.237,Z 1089.204,A -85,B 0,C 180,E1 13698.183,E2 13698.183} C_VEL
LIN {X 0,Y 479.332,Z 1071.129,A -85,B 0,C 180,E1 13701.032,E2 13701.032} C_VEL
LIN {X 0,Y 480.541,Z 1047.816,A -85,B 0,C 180,E1 13703.516,E2 13703.516} C_VEL
LIN {X 0,Y 481.818,Z 1021.237,A -85,B 0,C 180,E1 13705.394,E2 13705.394} C_VEL
LIN {X 0,Y 482.549,Z 991.613,A -85,B 0,C 180,E1 13706.67,E2 13706.67} C_VEL
LIN {X 0,Y 482.127,Z 958.459,A -85,B 0,C 180,E1 13707.386,E2 13707.386} C_VEL
LIN {X 0,Y 474.398,Z 923.03,A -85,B 0,C 180,E1 13708.336,E2 13708.336} C_VEL
LIN {X 0,Y 473.944,Z 923.03,A -85,B 0,C 180,E1 13715.025,E2 13715.025} C_VEL
LIN {X 0,Y 473.809,Z 923.03,A -85,B 0,C 180,E1 13722.05,E2 13722.05} C_VEL
LIN {X 0,Y 473.815,Z 923.03,A -85,B 0,C 180,E1 13727.937,E2 13727.937} C_VEL
LIN {X 0,Y 473.942,Z 923.03,A -85,B 0,C 180,E1 13732.856,E2 13732.856} C_VEL
LIN {X 0,Y 474.106,Z 923.03,A -85,B 0,C 180,E1 13739.383,E2 13739.383} C_VEL
LIN {X 0,Y 474.32,Z 923.03,A -85,B 0,C 180,E1 13745.519,E2 13745.519} C_VEL
LIN {X 0,Y 474.54,Z 923.03,A -85,B 0,C 180,E1 13751.417,E2 13751.417} C_VEL
LIN {X 0,Y 474.724,Z 923.03,A -85,B 0,C 180,E1 13757.11,E2 13757.11} C_VEL
LIN {X 0,Y 475.06,Z 923.03,A -85,B 0,C 180,E1 13762.675,E2 13762.675} C_VEL
LIN {X 0,Y 475.392,Z 923.03,A -85,B 0,C 180,E1 13768.163,E2 13768.163} C_VEL
LIN {X 0,Y 475.278,Z 923.03,A -85,B 0,C 180,E1 13773.629,E2 13773.629} C_VEL
LIN {X 0,Y 474.962,Z 923.03,A -85,B 0,C 180,E1 13779.494,E2 13779.494} C_VEL
LIN {X 0,Y 474.728,Z 923.03,A -85,B 0,C 180,E1 13784.735,E2 13784.735} C_VEL
LIN {X 0,Y 474.481,Z 923.03,A -85,B 0,C 180,E1 13790.488,E2 13790.488} C_VEL
LIN {X 0,Y 474.215,Z 923.03,A -85,B 0,C 180,E1 13796.841,E2 13796.841} C_VEL
LIN {X 0,Y 474.033,Z 923.03,A -85,B 0,C 180,E1 13802.792,E2 13802.792} C_VEL
LIN {X 0,Y 473.967,Z 923.03,A -85,B 0,C 180,E1 13807.259,E2 13807.259} C_VEL
LIN {X 0,Y 473.895,Z 923.03,A -85,B 0,C 180,E1 13812.825,E2 13812.825} C_VEL
LIN {X 0,Y 473.888,Z 923.03,A -85,B 0,C 180,E1 13817.959,E2 13817.959} C_VEL
LIN {X 0,Y 474.075,Z 923.498,A -85,B 0,C 180,E1 13824.323,E2 13824.323} C_VEL
LIN {X 0,Y 489.446,Z 966.149,A -85,B 0,C 180,E1 13826.525,E2 13826.525} C_VEL
LIN {X 0,Y 498.113,Z 996.728,A -85,B 0,C 180,E1 13828.394,E2 13828.394} C_VEL
LIN {X 0,Y 493.797,Z 1035.244,A -85,B 0,C 180,E1 13830.585,E2 13830.585} C_VEL
LIN {X 0,Y 489.065,Z 1071.41,A -85,B 0,C 180,E1 13833.479,E2 13833.479} C_VEL
LIN {X 0,Y 484.758,Z 1101.697,A -85,B 0,C 180,E1 13836.743,E2 13836.743} C_VEL
LIN {X 0,Y 481.214,Z 1126.923,A -85,B 0,C 180,E1 13840.337,E2 13840.337} C_VEL
LIN {X 0,Y 478.521,Z 1148.507,A -85,B 0,C 180,E1 13844.467,E2 13844.467} C_VEL
LIN {X 0,Y 476.931,Z 1164.01,A -85,B 0,C 180,E1 13848.577,E2 13848.577} C_VEL
LIN {X 0,Y 475.992,Z 1175.176,A -85,B 0,C 180,E1 13853.024,E2 13853.024} C_VEL
LIN {X 0,Y 475.735,Z 1180.083,A -85,B 0,C 180,E1 13856.356,E2 13856.356} C_VEL
LIN {X 0,Y 475.62,Z 1182.3,A -85,B 0,C 180,E1 13859.998,E2 13859.998} C_VEL
LIN {X 0,Y 475.814,Z 1181.184,A -85,B 0,C 180,E1 13863.64,E2 13863.64} C_VEL
LIN {X 0,Y 476.52,Z 1175.118,A -85,B 0,C 180,E1 13868.202,E2 13868.202} C_VEL
LIN {X 0,Y 477.823,Z 1163.54,A -85,B 0,C 180,E1 13872.788,E2 13872.788} C_VEL
LIN {X 0,Y 480.252,Z 1146.772,A -85,B 0,C 180,E1 13877.154,E2 13877.154} C_VEL
LIN {X 0,Y 484.016,Z 1124.581,A -85,B 0,C 180,E1 13881.278,E2 13881.278} C_VEL
LIN {X 0,Y 488.654,Z 1098.195,A -85,B 0,C 180,E1 13884.917,E2 13884.917} C_VEL
LIN {X 0,Y 494.21,Z 1066.678,A -85,B 0,C 180,E1 13888.163,E2 13888.163} C_VEL
LIN {X 0,Y 500.106,Z 1028.9,A -85,B 0,C 180,E1 13891.032,E2 13891.032} C_VEL
LIN {X 0,Y 503.959,Z 995.744,A -85,B 0,C 180,E1 13892.942,E2 13892.942} C_VEL
LIN {X 0,Y 498.944,Z 971.293,A -85,B 0,C 180,E1 13894.911,E2 13894.911} C_VEL
LIN {X 0,Y 491.362,Z 952.424,A -85,B 0,C 180,E1 13897.024,E2 13897.024} C_VEL
LIN {X 0,Y 485.078,Z 941.475,A -85,B 0,C 180,E1 13898.882,E2 13898.882} C_VEL
LIN {X 0,Y 481.914,Z 936.226,A -85,B 0,C 180,E1 13900.08,E2 13900.08} C_VEL
LIN {X 0,Y 478.599,Z 930.21,A -85,B 0,C 180,E1 13901.987,E2 13901.987} C_VEL
LIN {X 0,Y 476.691,Z 929.146,A -85,B 0,C 180,E1 13905.047,E2 13905.047} C_VEL
LIN {X 0,Y 479.309,Z 931.318,A -85,B 0,C 180,E1 13907.509,E2 13907.509} C_VEL
LIN {X 0,Y 483.936,Z 939.264,A -85,B 0,C 180,E1 13909.721,E2 13909.721} C_VEL
LIN {X 0,Y 489.977,Z 949.237,A -85,B 0,C 180,E1 13911.577,E2 13911.577} C_VEL
LIN {X 0,Y 498.631,Z 967.337,A -85,B 0,C 180,E1 13913.692,E2 13913.692} C_VEL
LIN {X 0,Y 505.425,Z 989.657,A -85,B 0,C 180,E1 13915.407,E2 13915.407} C_VEL
LIN {X 0,Y 505.944,Z 998.574,A -85,B 0,C 180,E1 13915.849,E2 13915.849} C_VEL
LIN {X 0,Y 500.213,Z 1041.859,A -85,B 0,C 180,E1 13917.651,E2 13917.651} C_VEL
LIN {X 0,Y 494.215,Z 1082.358,A -85,B 0,C 180,E1 13920.102,E2 13920.102} C_VEL
LIN {X 0,Y 488.514,Z 1119.918,A -85,B 0,C 180,E1 13923.248,E2 13923.248} C_VEL
LIN {X 0,Y 483.576,Z 1151.817,A -85,B 0,C 180,E1 13926.856,E2 13926.856} C_VEL
LIN {X 0,Y 479.767,Z 1178.475,A -85,B 0,C 180,E1 13930.884,E2 13930.884} C_VEL
LIN {X 0,Y 477.475,Z 1198.418,A -85,B 0,C 180,E1 13934.942,E2 13934.942} C_VEL
LIN {X 0,Y 476.284,Z 1213.001,A -85,B 0,C 180,E1 13939.043,E2 13939.043} C_VEL
LIN {X 0,Y 476.126,Z 1215.22,A -85,B 0,C 180,E1 13939.846,E2 13939.846} C_VEL
LIN {X 0,Y 474.776,Z 1217.814,A -85,B 0,C 180,E1 13940.84,E2 13940.84} C_VEL
LIN {X 0,Y 468.028,Z 1223.256,A -85,B 0,C 180,E1 13943.599,E2 13943.599} C_VEL
LIN {X 0,Y 467.914,Z 1223.641,A -85,B 0,C 180,E1 13943.864,E2 13943.864} C_VEL
LIN {X 0,Y 467.828,Z 1227.922,A -85,B 0,C 180,E1 13948.165,E2 13948.165} C_VEL
LIN {X 0,Y 467.921,Z 1227.723,A -85,B 0,C 180,E1 13951.867,E2 13951.867} C_VEL
LIN {X 0,Y 467.96,Z 1222.519,A -85,B 0,C 180,E1 13956.505,E2 13956.505} C_VEL
LIN {X 0,Y 468.282,Z 1213.47,A -85,B 0,C 180,E1 13960.519,E2 13960.519} C_VEL
LIN {X 0,Y 469.517,Z 1197.4,A -85,B 0,C 180,E1 13965.097,E2 13965.097} C_VEL
LIN {X 0,Y 471.892,Z 1175.975,A -85,B 0,C 180,E1 13969.382,E2 13969.382} C_VEL
LIN {X 0,Y 475.445,Z 1150.068,A -85,B 0,C 180,E1 13973.213,E2 13973.213} C_VEL
LIN {X 0,Y 479.714,Z 1120.032,A -85,B 0,C 180,E1 13976.56,E2 13976.56} C_VEL
LIN {X 0,Y 484.417,Z 1086.274,A -85,B 0,C 180,E1 13979.379,E2 13979.379} C_VEL
LIN {X 0,Y 489.115,Z 1048.101,A -85,B 0,C 180,E1 13981.697,E2 13981.697} C_VEL
LIN {X 0,Y 493.254,Z 1006.084,A -85,B 0,C 180,E1 13983.407,E2 13983.407} C_VEL
LIN {X 0,Y 493.18,Z 994.187,A -85,B 0,C 180,E1 13983.811,E2 13983.811} C_VEL
LIN {X 0,Y 468.74,Z 930.872,A -85,B 0,C 180,E1 13986.762,E2 13986.762} C_VEL
LIN {X 0,Y 466.109,Z 923.03,A -85,B 0,C 180,E1 13987.15,E2 13987.15} C_VEL
LIN {X 0,Y 465.908,Z 923.03,A -85,B 0,C 180,E1 13992.947,E2 13992.947} C_VEL
LIN {X 0,Y 465.897,Z 923.03,A -85,B 0,C 180,E1 13999.56,E2 13999.56} C_VEL
LIN {X 0,Y 466.014,Z 923.03,A -85,B 0,C 180,E1 14006.55,E2 14006.55} C_VEL
LIN {X 0,Y 466.26,Z 923.03,A -85,B 0,C 180,E1 14013.019,E2 14013.019} C_VEL
LIN {X 0,Y 466.4,Z 923.03,A -85,B 0,C 180,E1 14019.123,E2 14019.123} C_VEL
LIN {X 0,Y 466.599,Z 923.03,A -85,B 0,C 180,E1 14024.986,E2 14024.986} C_VEL
LIN {X 0,Y 466.849,Z 923.03,A -85,B 0,C 180,E1 14028.626,E2 14028.626} C_VEL
LIN {X 0,Y 478.559,Z 957.198,A -85,B 0,C 180,E1 14030.238,E2 14030.238} C_VEL
LIN {X 0,Y 480.425,Z 967.806,A -85,B 0,C 180,E1 14030.581,E2 14030.581} C_VEL
LIN {X 0,Y 479.733,Z 1004.515,A -85,B 0,C 180,E1 14031.511,E2 14031.511} C_VEL
LIN {X 0,Y 478.438,Z 1033.84,A -85,B 0,C 180,E1 14032.972,E2 14032.972} C_VEL
LIN {X 0,Y 476.53,Z 1058.932,A -85,B 0,C 180,E1 14034.999,E2 14034.999} C_VEL
LIN {X 0,Y 474.51,Z 1079.447,A -85,B 0,C 180,E1 14037.492,E2 14037.492} C_VEL
LIN {X 0,Y 472.498,Z 1095.834,A -85,B 0,C 180,E1 14040.46,E2 14040.46} C_VEL
LIN {X 0,Y 470.898,Z 1106.74,A -85,B 0,C 180,E1 14043.682,E2 14043.682} C_VEL
LIN {X 0,Y 470.242,Z 1110.38,A -85,B 0,C 180,E1 14045.534,E2 14045.534} C_VEL
LIN {X 0,Y 469.754,Z 1112.364,A -85,B 0,C 180,E1 14047.395,E2 14047.395} C_VEL
LIN {X 0,Y 469.495,Z 1112.687,A -85,B 0,C 180,E1 14049.263,E2 14049.263} C_VEL
LIN {X 0,Y 469.477,Z 1109.995,A -85,B 0,C 180,E1 14052.078,E2 14052.078} C_VEL
LIN {X 0,Y 469.818,Z 1101.845,A -85,B 0,C 180,E1 14055.416,E2 14055.416} C_VEL
LIN {X 0,Y 470.572,Z 1087.395,A -85,B 0,C 180,E1 14058.733,E2 14058.733} C_VEL
LIN {X 0,Y 471.702,Z 1068.334,A -85,B 0,C 180,E1 14061.584,E2 14061.584} C_VEL
LIN {X 0,Y 473.041,Z 1043.911,A -85,B 0,C 180,E1 14064.037,E2 14064.037} C_VEL
LIN {X 0,Y 474.265,Z 1016.272,A -85,B 0,C 180,E1 14065.858,E2 14065.858} C_VEL
LIN {X 0,Y 474.928,Z 985.749,A -85,B 0,C 180,E1 14067.032,E2 14067.032} C_VEL
LIN {X 0,Y 474.263,Z 958.905,A -85,B 0,C 180,E1 14067.586,E2 14067.586} C_VEL
LIN {X 0,Y 466.453,Z 923.03,A -85,B 0,C 180,E1 14068.535,E2 14068.535} C_VEL
LIN {X 0,Y 465.956,Z 923.03,A -85,B 0,C 180,E1 14075.81,E2 14075.81} C_VEL
LIN {X 0,Y 465.904,Z 923.03,A -85,B 0,C 180,E1 14081.739,E2 14081.739} C_VEL
LIN {X 0,Y 465.915,Z 923.03,A -85,B 0,C 180,E1 14088.244,E2 14088.244} C_VEL
LIN {X 0,Y 465.974,Z 923.03,A -85,B 0,C 180,E1 14094.271,E2 14094.271} C_VEL
LIN {X 0,Y 466.262,Z 923.03,A -85,B 0,C 180,E1 14101.053,E2 14101.053} C_VEL
LIN {X 0,Y 466.425,Z 923.03,A -85,B 0,C 180,E1 14107.107,E2 14107.107} C_VEL
LIN {X 0,Y 466.696,Z 923.03,A -85,B 0,C 180,E1 14113.042,E2 14113.042} C_VEL
LIN {X 0,Y 466.89,Z 923.03,A -85,B 0,C 180,E1 14118.787,E2 14118.787} C_VEL
LIN {X 0,Y 467.292,Z 923.03,A -85,B 0,C 180,E1 14124.417,E2 14124.417} C_VEL
LIN {X 0,Y 467.678,Z 923.03,A -85,B 0,C 180,E1 14129.984,E2 14129.984} C_VEL
LIN {X 0,Y 467.344,Z 923.03,A -85,B 0,C 180,E1 14135.55,E2 14135.55} C_VEL
LIN {X 0,Y 466.965,Z 923.03,A -85,B 0,C 180,E1 14141.178,E2 14141.178} C_VEL
LIN {X 0,Y 466.751,Z 923.03,A -85,B 0,C 180,E1 14146.921,E2 14146.921} C_VEL
LIN {X 0,Y 466.429,Z 923.03,A -85,B 0,C 180,E1 14152.858,E2 14152.858} C_VEL
LIN {X 0,Y 466.248,Z 923.03,A -85,B 0,C 180,E1 14159.066,E2 14159.066} C_VEL
LIN {X 0,Y 466.029,Z 923.03,A -85,B 0,C 180,E1 14165.684,E2 14165.684} C_VEL
LIN {X 0,Y 465.988,Z 923.03,A -85,B 0,C 180,E1 14171.766,E2 14171.766} C_VEL
LIN {X 0,Y 465.971,Z 923.03,A -85,B 0,C 180,E1 14178.203,E2 14178.203} C_VEL
LIN {X 0,Y 466.104,Z 923.071,A -85,B 0,C 180,E1 14183.813,E2 14183.813} C_VEL
LIN {X 0,Y 481.61,Z 966.314,A -85,B 0,C 180,E1 14186.081,E2 14186.081} C_VEL
LIN {X 0,Y 490.792,Z 998.091,A -85,B 0,C 180,E1 14188.074,E2 14188.074} C_VEL
LIN {X 0,Y 486.123,Z 1038.058,A -85,B 0,C 180,E1 14190.42,E2 14190.42} C_VEL
LIN {X 0,Y 481.5,Z 1072.313,A -85,B 0,C 180,E1 14193.231,E2 14193.231} C_VEL
LIN {X 0,Y 477.152,Z 1102.128,A -85,B 0,C 180,E1 14196.496,E2 14196.496} C_VEL
LIN {X 0,Y 473.492,Z 1127.468,A -85,B 0,C 180,E1 14200.164,E2 14200.164} C_VEL
LIN {X 0,Y 470.746,Z 1148.727,A -85,B 0,C 180,E1 14204.287,E2 14204.287} C_VEL
LIN {X 0,Y 469.084,Z 1164.071,A -85,B 0,C 180,E1 14208.383,E2 14208.383} C_VEL
LIN {X 0,Y 468.101,Z 1175.576,A -85,B 0,C 180,E1 14213.007,E2 14213.007} C_VEL
LIN {X 0,Y 467.859,Z 1180.396,A -85,B 0,C 180,E1 14216.294,E2 14216.294} C_VEL
LIN {X 0,Y 467.745,Z 1182.693,A -85,B 0,C 180,E1 14219.998,E2 14219.998} C_VEL
LIN {X 0,Y 467.949,Z 1181.678,A -85,B 0,C 180,E1 14223.701,E2 14223.701} C_VEL
LIN {X 0,Y 468.681,Z 1175.707,A -85,B 0,C 180,E1 14228.34,E2 14228.34} C_VEL
LIN {X 0,Y 470.081,Z 1164.229,A -85,B 0,C 180,E1 14233.002,E2 14233.002} C_VEL
LIN {X 0,Y 472.675,Z 1147.574,A -85,B 0,C 180,E1 14237.438,E2 14237.438} C_VEL
LIN {X 0,Y 476.683,Z 1125.535,A -85,B 0,C 180,E1 14241.622,E2 14241.622} C_VEL
LIN {X 0,Y 481.579,Z 1099.386,A -85,B 0,C 180,E1 14245.308,E2 14245.308} C_VEL
LIN {X 0,Y 487.403,Z 1068.246,A -85,B 0,C 180,E1 14248.592,E2 14248.592} C_VEL
LIN {X 0,Y 493.594,Z 1031.514,A -85,B 0,C 180,E1 14251.468,E2 14251.468} C_VEL
LIN {X 0,Y 497.925,Z 998.931,A -85,B 0,C 180,E1 14253.393,E2 14253.393} C_VEL
LIN {X 0,Y 493.59,Z 975.28,A -85,B 0,C 180,E1 14255.4,E2 14255.4} C_VEL
LIN {X 0,Y 486.541,Z 956.903,A -85,B 0,C 180,E1 14257.615,E2 14257.615} C_VEL
LIN {X 0,Y 479.871,Z 944.014,A -85,B 0,C 180,E1 14260.059,E2 14260.059} C_VEL
LIN {X 0,Y 476.338,Z 937.757,A -85,B 0,C 180,E1 14262.121,E2 14262.121} C_VEL
LIN {X 0,Y 474.661,Z 936.79,A -85,B 0,C 180,E1 14265.082,E2 14265.082} C_VEL
LIN {X 0,Y 476.83,Z 938.817,A -85,B 0,C 180,E1 14267.287,E2 14267.287} C_VEL
LIN {X 0,Y 481.169,Z 946.63,A -85,B 0,C 180,E1 14269.516,E2 14269.516} C_VEL
LIN {X 0,Y 487.08,Z 957.22,A -85,B 0,C 180,E1 14271.442,E2 14271.442} C_VEL
LIN {X 0,Y 494.645,Z 974.467,A -85,B 0,C 180,E1 14273.461,E2 14273.461} C_VEL
LIN {X 0,Y 500.208,Z 996.684,A -85,B 0,C 180,E1 14275.164,E2 14275.164} C_VEL
LIN {X 0,Y 494.071,Z 1040.852,A -85,B 0,C 180,E1 14277.037,E2 14277.037} C_VEL
LIN {X 0,Y 487.679,Z 1081.455,A -85,B 0,C 180,E1 14279.531,E2 14279.531} C_VEL
LIN {X 0,Y 481.579,Z 1118.918,A -85,B 0,C 180,E1 14282.704,E2 14282.704} C_VEL
LIN {X 0,Y 476.394,Z 1150.622,A -85,B 0,C 180,E1 14286.327,E2 14286.327} C_VEL
LIN {X 0,Y 472.423,Z 1176.714,A -85,B 0,C 180,E1 14290.287,E2 14290.287} C_VEL
LIN {X 0,Y 469.753,Z 1197.664,A -85,B 0,C 180,E1 14294.57,E2 14294.57} C_VEL
LIN {X 0,Y 468.41,Z 1212.674,A -85,B 0,C 180,E1 14298.857,E2 14298.857} C_VEL
LIN {X 0,Y 467.952,Z 1223.139,A -85,B 0,C 180,E1 14303.528,E2 14303.528} C_VEL
LIN {X 0,Y 467.914,Z 1223.641,A -85,B 0,C 180,E1 14303.864,E2 14303.864} C_VEL
LIN {X 0,Y 465.282,Z 1225.683,A -85,B 0,C 180,E1 14305.425,E2 14305.425} C_VEL
LIN {X 0,Y 459.99,Z 1227.391,A -85,B 0,C 180,E1 14307.788,E2 14307.788} C_VEL
LIN {X 0,Y 459.925,Z 1227.471,A -85,B 0,C 180,E1 14308.061,E2 14308.061} C_VEL
LIN {X 0,Y 460.026,Z 1227.271,A -85,B 0,C 180,E1 14311.899,E2 14311.899} C_VEL
LIN {X 0,Y 460.089,Z 1221.969,A -85,B 0,C 180,E1 14316.617,E2 14316.617} C_VEL
LIN {X 0,Y 460.47,Z 1211.937,A -85,B 0,C 180,E1 14320.986,E2 14320.986} C_VEL
LIN {X 0,Y 461.726,Z 1196.53,A -85,B 0,C 180,E1 14325.358,E2 14325.358} C_VEL
LIN {X 0,Y 464.2,Z 1175.201,A -85,B 0,C 180,E1 14329.658,E2 14329.658} C_VEL
LIN {X 0,Y 467.895,Z 1148.93,A -85,B 0,C 180,E1 14333.572,E2 14333.572} C_VEL
LIN {X 0,Y 472.379,Z 1118.248,A -85,B 0,C 180,E1 14337.006,E2 14337.006} C_VEL
LIN {X 0,Y 477.448,Z 1083.135,A -85,B 0,C 180,E1 14339.926,E2 14339.926} C_VEL
LIN {X 0,Y 482.462,Z 1043.162,A -85,B 0,C 180,E1 14342.3,E2 14342.3} C_VEL
LIN {X 0,Y 486.262,Z 1003.523,A -85,B 0,C 180,E1 14343.877,E2 14343.877} C_VEL
LIN {X 0,Y 485.577,Z 995.019,A -85,B 0,C 180,E1 14344.21,E2 14344.21} C_VEL
LIN {X 0,Y 462.179,Z 934.302,A -85,B 0,C 180,E1 14347.108,E2 14347.108} C_VEL
LIN {X 0,Y 458.099,Z 923.03,A -85,B 0,C 180,E1 14347.661,E2 14347.661} C_VEL
LIN {X 0,Y 457.971,Z 923.03,A -85,B 0,C 180,E1 14353.878,E2 14353.878} C_VEL
LIN {X 0,Y 458.015,Z 923.03,A -85,B 0,C 180,E1 14359.38,E2 14359.38} C_VEL
LIN {X 0,Y 458.029,Z 923.03,A -85,B 0,C 180,E1 14365.888,E2 14365.888} C_VEL
LIN {X 0,Y 458.311,Z 923.03,A -85,B 0,C 180,E1 14372.512,E2 14372.512} C_VEL
LIN {X 0,Y 458.446,Z 923.03,A -85,B 0,C 180,E1 14378.744,E2 14378.744} C_VEL
LIN {X 0,Y 458.651,Z 923.03,A -85,B 0,C 180,E1 14384.72,E2 14384.72} C_VEL
LIN {X 0,Y 458.937,Z 923.531,A -85,B 0,C 180,E1 14388.076,E2 14388.076} C_VEL
LIN {X 0,Y 471.257,Z 957.823,A -85,B 0,C 180,E1 14389.791,E2 14389.791} C_VEL
LIN {X 0,Y 473.315,Z 969.809,A -85,B 0,C 180,E1 14390.192,E2 14390.192} C_VEL
LIN {X 0,Y 472.595,Z 1006.339,A -85,B 0,C 180,E1 14391.15,E2 14391.15} C_VEL
LIN {X 0,Y 471.184,Z 1035.184,A -85,B 0,C 180,E1 14392.632,E2 14392.632} C_VEL
LIN {X 0,Y 469.16,Z 1060.171,A -85,B 0,C 180,E1 14394.689,E2 14394.689} C_VEL
LIN {X 0,Y 467.039,Z 1080.661,A -85,B 0,C 180,E1 14397.22,E2 14397.22} C_VEL
LIN {X 0,Y 464.897,Z 1096.939,A -85,B 0,C 180,E1 14400.235,E2 14400.235} C_VEL
LIN {X 0,Y 463.28,Z 1107.234,A -85,B 0,C 180,E1 14403.274,E2 14403.274} C_VEL
LIN {X 0,Y 462.414,Z 1111.782,A -85,B 0,C 180,E1 14405.628,E2 14405.628} C_VEL
LIN {X 0,Y 461.9,Z 1113.525,A -85,B 0,C 180,E1 14407.521,E2 14407.521} C_VEL
LIN {X 0,Y 461.632,Z 1112.562,A -85,B 0,C 180,E1 14410.823,E2 14410.823} C_VEL
LIN {X 0,Y 461.824,Z 1106.333,A -85,B 0,C 180,E1 14414.208,E2 14414.208} C_VEL
LIN {X 0,Y 462.346,Z 1094.63,A -85,B 0,C 180,E1 14417.503,E2 14417.503} C_VEL
LIN {X 0,Y 463.355,Z 1077.726,A -85,B 0,C 180,E1 14420.525,E2 14420.525} C_VEL
LIN {X 0,Y 464.732,Z 1054.619,A -85,B 0,C 180,E1 14423.282,E2 14423.282} C_VEL
LIN {X 0,Y 466.011,Z 1029.063,A -85,B 0,C 180,E1 14425.319,E2 14425.319} C_VEL
LIN {X 0,Y 466.975,Z 999.252,A -85,B 0,C 180,E1 14426.811,E2 14426.811} C_VEL
LIN {X 0,Y 466.971,Z 961.831,A -85,B 0,C 180,E1 14427.725,E2 14427.725} C_VEL
LIN {X 0,Y 458.499,Z 923.03,A -85,B 0,C 180,E1 14428.769,E2 14428.769} C_VEL
LIN {X 0,Y 458.019,Z 923.03,A -85,B 0,C 180,E1 14434.41,E2 14434.41} C_VEL
LIN {X 0,Y 457.988,Z 923.03,A -85,B 0,C 180,E1 14441.294,E2 14441.294} C_VEL
LIN {X 0,Y 457.996,Z 923.03,A -85,B 0,C 180,E1 14446.543,E2 14446.543} C_VEL
LIN {X 0,Y 458.009,Z 923.03,A -85,B 0,C 180,E1 14452.36,E2 14452.36} C_VEL
LIN {X 0,Y 458.199,Z 923.03,A -85,B 0,C 180,E1 14459.036,E2 14459.036} C_VEL
LIN {X 0,Y 458.416,Z 923.03,A -85,B 0,C 180,E1 14464.61,E2 14464.61} C_VEL
LIN {X 0,Y 458.651,Z 923.03,A -85,B 0,C 180,E1 14470.748,E2 14470.748} C_VEL
LIN {X 0,Y 458.896,Z 923.03,A -85,B 0,C 180,E1 14476.658,E2 14476.658} C_VEL
LIN {X 0,Y 459.234,Z 923.03,A -85,B 0,C 180,E1 14482.421,E2 14482.421} C_VEL
LIN {X 0,Y 459.597,Z 923.03,A -85,B 0,C 180,E1 14488.099,E2 14488.099} C_VEL
LIN {X 0,Y 459.461,Z 923.03,A -85,B 0,C 180,E1 14493.754,E2 14493.754} C_VEL
LIN {X 0,Y 459.156,Z 923.03,A -85,B 0,C 180,E1 14499.453,E2 14499.453} C_VEL
LIN {X 0,Y 458.85,Z 923.03,A -85,B 0,C 180,E1 14505.257,E2 14505.257} C_VEL
LIN {X 0,Y 458.565,Z 923.03,A -85,B 0,C 180,E1 14511.233,E2 14511.233} C_VEL
LIN {X 0,Y 458.365,Z 923.03,A -85,B 0,C 180,E1 14517.465,E2 14517.465} C_VEL
LIN {X 0,Y 458.108,Z 923.03,A -85,B 0,C 180,E1 14524.084,E2 14524.084} C_VEL
LIN {X 0,Y 458.059,Z 923.03,A -85,B 0,C 180,E1 14530.643,E2 14530.643} C_VEL
LIN {X 0,Y 458.058,Z 923.03,A -85,B 0,C 180,E1 14536.502,E2 14536.502} C_VEL
LIN {X 0,Y 458.184,Z 923.03,A -85,B 0,C 180,E1 14543.291,E2 14543.291} C_VEL
LIN {X 0,Y 474.03,Z 967.377,A -85,B 0,C 180,E1 14545.679,E2 14545.679} C_VEL
LIN {X 0,Y 483.416,Z 999.681,A -85,B 0,C 180,E1 14547.757,E2 14547.757} C_VEL
LIN {X 0,Y 478.596,Z 1039.511,A -85,B 0,C 180,E1 14550.159,E2 14550.159} C_VEL
LIN {X 0,Y 473.737,Z 1074.647,A -85,B 0,C 180,E1 14553.125,E2 14553.125} C_VEL
LIN {X 0,Y 469.293,Z 1104.203,A -85,B 0,C 180,E1 14556.463,E2 14556.463} C_VEL
LIN {X 0,Y 465.417,Z 1130.2,A -85,B 0,C 180,E1 14560.364,E2 14560.364} C_VEL
LIN {X 0,Y 462.787,Z 1150.354,A -85,B 0,C 180,E1 14564.433,E2 14564.433} C_VEL
LIN {X 0,Y 460.973,Z 1167.092,A -85,B 0,C 180,E1 14569.186,E2 14569.186} C_VEL
LIN {X 0,Y 460.189,Z 1176.697,A -85,B 0,C 180,E1 14573.399,E2 14573.399} C_VEL
LIN {X 0,Y 459.957,Z 1182.3,A -85,B 0,C 180,E1 14578.115,E2 14578.115} C_VEL
LIN {X 0,Y 459.966,Z 1183.06,A -85,B 0,C 180,E1 14581.881,E2 14581.881} C_VEL
LIN {X 0,Y 460.477,Z 1179.268,A -85,B 0,C 180,E1 14586.593,E2 14586.593} C_VEL
LIN {X 0,Y 461.595,Z 1170.179,A -85,B 0,C 180,E1 14591.326,E2 14591.326} C_VEL
LIN {X 0,Y 464.083,Z 1154.69,A -85,B 0,C 180,E1 14596.208,E2 14596.208} C_VEL
LIN {X 0,Y 467.671,Z 1134.988,A -85,B 0,C 180,E1 14600.504,E2 14600.504} C_VEL
LIN {X 0,Y 472.759,Z 1109.558,A -85,B 0,C 180,E1 14604.55,E2 14604.55} C_VEL
LIN {X 0,Y 478.672,Z 1080.136,A -85,B 0,C 180,E1 14608.037,E2 14608.037} C_VEL
LIN {X 0,Y 485.292,Z 1044.966,A -85,B 0,C 180,E1 14611.142,E2 14611.142} C_VEL
LIN {X 0,Y 491.799,Z 1005.476,A -85,B 0,C 180,E1 14613.654,E2 14613.654} C_VEL
LIN {X 0,Y 490.091,Z 987.044,A -85,B 0,C 180,E1 14615.149,E2 14615.149} C_VEL
LIN {X 0,Y 484.693,Z 967.993,A -85,B 0,C 180,E1 14617.243,E2 14617.243} C_VEL
LIN {X 0,Y 478.867,Z 955.211,A -85,B 0,C 180,E1 14619.432,E2 14619.432} C_VEL
LIN {X 0,Y 475.527,Z 949.289,A -85,B 0,C 180,E1 14621.02,E2 14621.02} C_VEL
LIN {X 0,Y 473.804,Z 945.149,A -85,B 0,C 180,E1 14622.462,E2 14622.462} C_VEL
LIN {X 0,Y 473.064,Z 944.712,A -85,B 0,C 180,E1 14625.834,E2 14625.834} C_VEL
LIN {X 0,Y 474.476,Z 946.558,A -85,B 0,C 180,E1 14627.146,E2 14627.146} C_VEL
LIN {X 0,Y 478.589,Z 954.287,A -85,B 0,C 180,E1 14629.374,E2 14629.374} C_VEL
LIN {X 0,Y 484.632,Z 966.071,A -85,B 0,C 180,E1 14631.467,E2 14631.467} C_VEL
LIN {X 0,Y 491.398,Z 984.719,A -85,B 0,C 180,E1 14633.504,E2 14633.504} C_VEL
LIN {X 0,Y 494.256,Z 999.78,A -85,B 0,C 180,E1 14634.644,E2 14634.644} C_VEL
LIN {X 0,Y 487.578,Z 1042.922,A -85,B 0,C 180,E1 14636.553,E2 14636.553} C_VEL
LIN {X 0,Y 480.645,Z 1083.889,A -85,B 0,C 180,E1 14639.168,E2 14639.168} C_VEL
LIN {X 0,Y 474.084,Z 1121.431,A -85,B 0,C 180,E1 14642.493,E2 14642.493} C_VEL
LIN {X 0,Y 468.947,Z 1151.213,A -85,B 0,C 180,E1 14646.015,E2 14646.015} C_VEL
LIN {X 0,Y 464.779,Z 1176.905,A -85,B 0,C 180,E1 14650.015,E2 14650.015} C_VEL
LIN {X 0,Y 462.008,Z 1197.132,A -85,B 0,C 180,E1 14654.231,E2 14654.231} C_VEL
LIN {X 0,Y 460.566,Z 1212.374,A -85,B 0,C 180,E1 14658.665,E2 14658.665} C_VEL
LIN {X 0,Y 460.044,Z 1222.792,A -85,B 0,C 180,E1 14663.416,E2 14663.416} C_VEL
LIN {X 0,Y 459.925,Z 1227.471,A -85,B 0,C 180,E1 14668.061,E2 14668.061} C_VEL
LIN {X 0,Y 457.546,Z 1227.858,A -85,B 0,C 180,E1 14669.666,E2 14669.666} C_VEL
LIN {X 0,Y 452.095,Z 1226.491,A -85,B 0,C 180,E1 14672.354,E2 14672.354} C_VEL
LIN {X 0,Y 452.207,Z 1221.395,A -85,B 0,C 180,E1 14676.733,E2 14676.733} C_VEL
LIN {X 0,Y 452.553,Z 1212.032,A -85,B 0,C 180,E1 14680.898,E2 14680.898} C_VEL
LIN {X 0,Y 453.861,Z 1196.309,A -85,B 0,C 180,E1 14685.463,E2 14685.463} C_VEL
LIN {X 0,Y 456.415,Z 1174.908,A -85,B 0,C 180,E1 14689.853,E2 14689.853} C_VEL
LIN {X 0,Y 460.14,Z 1149.346,A -85,B 0,C 180,E1 14693.737,E2 14693.737} C_VEL
LIN {X 0,Y 464.708,Z 1118.826,A -85,B 0,C 180,E1 14697.227,E2 14697.227} C_VEL
LIN {X 0,Y 469.88,Z 1083.963,A -85,B 0,C 180,E1 14700.191,E2 14700.191} C_VEL
LIN {X 0,Y 474.979,Z 1044.608,A -85,B 0,C 180,E1 14702.6,E2 14702.6} C_VEL
LIN {X 0,Y 479.218,Z 1002.134,A -85,B 0,C 180,E1 14704.315,E2 14704.315} C_VEL
LIN {X 0,Y 469.43,Z 972.203,A -85,B 0,C 180,E1 14705.781,E2 14705.781} C_VEL
LIN {X 0,Y 450.147,Z 923.03,A -85,B 0,C 180,E1 14708.295,E2 14708.295} C_VEL
LIN {X 0,Y 449.985,Z 923.03,A -85,B 0,C 180,E1 14715.157,E2 14715.157} C_VEL
LIN {X 0,Y 450.087,Z 923.03,A -85,B 0,C 180,E1 14720.571,E2 14720.571} C_VEL
LIN {X 0,Y 450.111,Z 923.03,A -85,B 0,C 180,E1 14727.088,E2 14727.088} C_VEL
LIN {X 0,Y 450.322,Z 923.03,A -85,B 0,C 180,E1 14731.982,E2 14731.982} C_VEL
LIN {X 0,Y 450.518,Z 923.03,A -85,B 0,C 180,E1 14738.351,E2 14738.351} C_VEL
LIN {X 0,Y 450.712,Z 923.03,A -85,B 0,C 180,E1 14744.444,E2 14744.444} C_VEL
LIN {X 0,Y 450.947,Z 923.643,A -85,B 0,C 180,E1 14747.432,E2 14747.432} C_VEL
LIN {X 0,Y 463.769,Z 957.498,A -85,B 0,C 180,E1 14749.276,E2 14749.276} C_VEL
LIN {X 0,Y 466.335,Z 969.99,A -85,B 0,C 180,E1 14749.745,E2 14749.745} C_VEL
LIN {X 0,Y 465.54,Z 1006.726,A -85,B 0,C 180,E1 14750.721,E2 14750.721} C_VEL
LIN {X 0,Y 464,Z 1036.718,A -85,B 0,C 180,E1 14752.282,E2 14752.282} C_VEL
LIN {X 0,Y 461.827,Z 1061.484,A -85,B 0,C 180,E1 14754.369,E2 14754.369} C_VEL
LIN {X 0,Y 459.38,Z 1083.4,A -85,B 0,C 180,E1 14757.174,E2 14757.174} C_VEL
LIN {X 0,Y 457.297,Z 1098.131,A -85,B 0,C 180,E1 14760.002,E2 14760.002} C_VEL
LIN {X 0,Y 455.49,Z 1108.897,A -85,B 0,C 180,E1 14763.33,E2 14763.33} C_VEL
LIN {X 0,Y 454.58,Z 1113.147,A -85,B 0,C 180,E1 14765.725,E2 14765.725} C_VEL
LIN {X 0,Y 454.048,Z 1114.615,A -85,B 0,C 180,E1 14767.652,E2 14767.652} C_VEL
LIN {X 0,Y 453.811,Z 1114.436,A -85,B 0,C 180,E1 14769.586,E2 14769.586} C_VEL
LIN {X 0,Y 453.837,Z 1109.945,A -85,B 0,C 180,E1 14772.99,E2 14772.99} C_VEL
LIN {X 0,Y 454.264,Z 1100.091,A -85,B 0,C 180,E1 14776.427,E2 14776.427} C_VEL
LIN {X 0,Y 455.189,Z 1084.639,A -85,B 0,C 180,E1 14779.643,E2 14779.643} C_VEL
LIN {X 0,Y 456.413,Z 1065.068,A -85,B 0,C 180,E1 14782.376,E2 14782.376} C_VEL
LIN {X 0,Y 457.685,Z 1040.271,A -85,B 0,C 180,E1 14784.733,E2 14784.733} C_VEL
LIN {X 0,Y 458.882,Z 1011.772,A -85,B 0,C 180,E1 14786.491,E2 14786.491} C_VEL
LIN {X 0,Y 459.55,Z 981.138,A -85,B 0,C 180,E1 14787.545,E2 14787.545} C_VEL
LIN {X 0,Y 458.676,Z 960.479,A -85,B 0,C 180,E1 14787.976,E2 14787.976} C_VEL
LIN {X 0,Y 450.564,Z 923.03,A -85,B 0,C 180,E1 14789.027,E2 14789.027} C_VEL
LIN {X 0,Y 450.082,Z 923.03,A -85,B 0,C 180,E1 14796.294,E2 14796.294} C_VEL
LIN {X 0,Y 450.01,Z 923.03,A -85,B 0,C 180,E1 14802.356,E2 14802.356} C_VEL
LIN {X 0,Y 450.032,Z 923.03,A -85,B 0,C 180,E1 14807.795,E2 14807.795} C_VEL
LIN {X 0,Y 450.1,Z 923.03,A -85,B 0,C 180,E1 14813.685,E2 14813.685} C_VEL
LIN {X 0,Y 450.322,Z 923.03,A -85,B 0,C 180,E1 14820.749,E2 14820.749} C_VEL
LIN {X 0,Y 450.523,Z 923.03,A -85,B 0,C 180,E1 14826.25,E2 14826.25} C_VEL
LIN {X 0,Y 450.806,Z 923.03,A -85,B 0,C 180,E1 14832.425,E2 14832.425} C_VEL
LIN {X 0,Y 451.043,Z 923.03,A -85,B 0,C 180,E1 14838.388,E2 14838.388} C_VEL
LIN {X 0,Y 451.451,Z 923.03,A -85,B 0,C 180,E1 14844.22,E2 14844.22} C_VEL
LIN {X 0,Y 451.886,Z 923.03,A -85,B 0,C 180,E1 14849.983,E2 14849.983} C_VEL
LIN {X 0,Y 451.5,Z 923.03,A -85,B 0,C 180,E1 14855.745,E2 14855.745} C_VEL
LIN {X 0,Y 451.112,Z 923.03,A -85,B 0,C 180,E1 14861.576,E2 14861.576} C_VEL
LIN {X 0,Y 450.852,Z 923.03,A -85,B 0,C 180,E1 14867.537,E2 14867.537} C_VEL
LIN {X 0,Y 450.504,Z 923.03,A -85,B 0,C 180,E1 14873.714,E2 14873.714} C_VEL
LIN {X 0,Y 450.349,Z 923.03,A -85,B 0,C 180,E1 14880.196,E2 14880.196} C_VEL
LIN {X 0,Y 450.134,Z 923.03,A -85,B 0,C 180,E1 14887.15,E2 14887.15} C_VEL
LIN {X 0,Y 450.078,Z 923.03,A -85,B 0,C 180,E1 14892.382,E2 14892.382} C_VEL
LIN {X 0,Y 450.066,Z 923.03,A -85,B 0,C 180,E1 14897.814,E2 14897.814} C_VEL
LIN {X 0,Y 450.196,Z 923.03,A -85,B 0,C 180,E1 14902.763,E2 14902.763} C_VEL
LIN {X 0,Y 466.132,Z 967.35,A -85,B 0,C 180,E1 14905.208,E2 14905.208} C_VEL
LIN {X 0,Y 476.088,Z 1000.943,A -85,B 0,C 180,E1 14907.424,E2 14907.424} C_VEL
LIN {X 0,Y 471.283,Z 1039.649,A -85,B 0,C 180,E1 14909.8,E2 14909.8} C_VEL
LIN {X 0,Y 466.461,Z 1073.541,A -85,B 0,C 180,E1 14912.675,E2 14912.675} C_VEL
LIN {X 0,Y 461.751,Z 1104.241,A -85,B 0,C 180,E1 14916.164,E2 14916.164} C_VEL
LIN {X 0,Y 457.793,Z 1129.988,A -85,B 0,C 180,E1 14920.064,E2 14920.064} C_VEL
LIN {X 0,Y 454.964,Z 1150.865,A -85,B 0,C 180,E1 14924.325,E2 14924.325} C_VEL
LIN {X 0,Y 453.172,Z 1166.771,A -85,B 0,C 180,E1 14928.875,E2 14928.875} C_VEL
LIN {X 0,Y 452.307,Z 1176.9,A -85,B 0,C 180,E1 14933.283,E2 14933.283} C_VEL
LIN {X 0,Y 452.092,Z 1182.648,A -85,B 0,C 180,E1 14938.083,E2 14938.083} C_VEL
LIN {X 0,Y 452.101,Z 1183.498,A -85,B 0,C 180,E1 14941.913,E2 14941.913} C_VEL
LIN {X 0,Y 452.639,Z 1179.827,A -85,B 0,C 180,E1 14946.708,E2 14946.708} C_VEL
LIN {X 0,Y 453.845,Z 1170.856,A -85,B 0,C 180,E1 14951.522,E2 14951.522} C_VEL
LIN {X 0,Y 456.347,Z 1156.302,A -85,B 0,C 180,E1 14956.282,E2 14956.282} C_VEL
LIN {X 0,Y 460.31,Z 1136.035,A -85,B 0,C 180,E1 14960.847,E2 14960.847} C_VEL
LIN {X 0,Y 465.698,Z 1110.874,A -85,B 0,C 180,E1 14964.948,E2 14964.948} C_VEL
LIN {X 0,Y 471.902,Z 1081.862,A -85,B 0,C 180,E1 14968.476,E2 14968.476} C_VEL
LIN {X 0,Y 478.802,Z 1047.551,A -85,B 0,C 180,E1 14971.596,E2 14971.596} C_VEL
LIN {X 0,Y 485.788,Z 1008.723,A -85,B 0,C 180,E1 14974.168,E2 14974.168} C_VEL
LIN {X 0,Y 485.088,Z 993.51,A -85,B 0,C 180,E1 14975.399,E2 14975.399} C_VEL
LIN {X 0,Y 480.889,Z 975.303,A -85,B 0,C 180,E1 14977.43,E2 14977.43} C_VEL
LIN {X 0,Y 475.605,Z 962.026,A -85,B 0,C 180,E1 14979.715,E2 14979.715} C_VEL
LIN {X 0,Y 472.36,Z 955.306,A -85,B 0,C 180,E1 14981.651,E2 14981.651} C_VEL
LIN {X 0,Y 471.324,Z 952.559,A -85,B 0,C 180,E1 14982.739,E2 14982.739} C_VEL
LIN {X 0,Y 471.16,Z 952.428,A -85,B 0,C 180,E1 14986.016,E2 14986.016} C_VEL
LIN {X 0,Y 472.223,Z 954.627,A -85,B 0,C 180,E1 14987.121,E2 14987.121} C_VEL
LIN {X 0,Y 475.94,Z 961.82,A -85,B 0,C 180,E1 14989.24,E2 14989.24} C_VEL
LIN {X 0,Y 481.897,Z 974.923,A -85,B 0,C 180,E1 14991.482,E2 14991.482} C_VEL
LIN {X 0,Y 487.408,Z 994.3,A -85,B 0,C 180,E1 14993.479,E2 14993.479} C_VEL
LIN {X 0,Y 488.162,Z 1003.534,A -85,B 0,C 180,E1 14994.112,E2 14994.112} C_VEL
LIN {X 0,Y 481.066,Z 1046.262,A -85,B 0,C 180,E1 14996.118,E2 14996.118} C_VEL
LIN {X 0,Y 473.424,Z 1087.764,A -85,B 0,C 180,E1 14998.912,E2 14998.912} C_VEL
LIN {X 0,Y 466.836,Z 1122.941,A -85,B 0,C 180,E1 15002.16,E2 15002.16} C_VEL
LIN {X 0,Y 461.293,Z 1153.023,A -85,B 0,C 180,E1 15005.849,E2 15005.849} C_VEL
LIN {X 0,Y 456.857,Z 1179.004,A -85,B 0,C 180,E1 15010.073,E2 15010.073} C_VEL
LIN {X 0,Y 453.819,Z 1200.73,A -85,B 0,C 180,E1 15014.925,E2 15014.925} C_VEL
LIN {X 0,Y 452.445,Z 1215.603,A -85,B 0,C 180,E1 15019.813,E2 15019.813} C_VEL
LIN {X 0,Y 452.094,Z 1223.854,A -85,B 0,C 180,E1 15024.263,E2 15024.263} C_VEL
LIN {X 0,Y 452.051,Z 1227.114,A -85,B 0,C 180,E1 15028.101,E2 15028.101} C_VEL
LIN {X 0,Y 452.095,Z 1226.491,A -85,B 0,C 180,E1 15032.354,E2 15032.354} C_VEL
LIN {X 0,Y 450.782,Z 1225.639,A -85,B 0,C 180,E1 15033.445,E2 15033.445} C_VEL
LIN {X 0,Y 444.359,Z 1221.566,A -85,B 0,C 180,E1 15036.403,E2 15036.403} C_VEL
LIN {X 0,Y 444.291,Z 1221.094,A -85,B 0,C 180,E1 15036.681,E2 15036.681} C_VEL
LIN {X 0,Y 444.729,Z 1210.745,A -85,B 0,C 180,E1 15041.283,E2 15041.283} C_VEL
LIN {X 0,Y 446.083,Z 1195.365,A -85,B 0,C 180,E1 15045.74,E2 15045.74} C_VEL
LIN {X 0,Y 448.78,Z 1173.705,A -85,B 0,C 180,E1 15050.206,E2 15050.206} C_VEL
LIN {X 0,Y 452.639,Z 1147.815,A -85,B 0,C 180,E1 15054.155,E2 15054.155} C_VEL
LIN {X 0,Y 457.404,Z 1116.918,A -85,B 0,C 180,E1 15057.699,E2 15057.699} C_VEL
LIN {X 0,Y 462.97,Z 1080.064,A -85,B 0,C 180,E1 15060.815,E2 15060.815} C_VEL
LIN {X 0,Y 468.061,Z 1041.786,A -85,B 0,C 180,E1 15063.11,E2 15063.11} C_VEL
LIN {X 0,Y 471.828,Z 1001.204,A -85,B 0,C 180,E1 15064.768,E2 15064.768} C_VEL
LIN {X 0,Y 454.496,Z 954.252,A -85,B 0,C 180,E1 15067.142,E2 15067.142} C_VEL
LIN {X 0,Y 442.237,Z 923.03,A -85,B 0,C 180,E1 15068.754,E2 15068.754} C_VEL
LIN {X 0,Y 442.014,Z 923.03,A -85,B 0,C 180,E1 15075.902,E2 15075.902} C_VEL
LIN {X 0,Y 442.116,Z 923.03,A -85,B 0,C 180,E1 15082.035,E2 15082.035} C_VEL
LIN {X 0,Y 442.241,Z 923.03,A -85,B 0,C 180,E1 15088.699,E2 15088.699} C_VEL
LIN {X 0,Y 442.441,Z 923.03,A -85,B 0,C 180,E1 15093.643,E2 15093.643} C_VEL
LIN {X 0,Y 442.642,Z 923.03,A -85,B 0,C 180,E1 15100.041,E2 15100.041} C_VEL
LIN {X 0,Y 442.976,Z 923.03,A -85,B 0,C 180,E1 15106.719,E2 15106.719} C_VEL
LIN {X 0,Y 456.738,Z 958.85,A -85,B 0,C 180,E1 15108.805,E2 15108.805} C_VEL
LIN {X 0,Y 459.355,Z 973.126,A -85,B 0,C 180,E1 15109.342,E2 15109.342} C_VEL
LIN {X 0,Y 458.469,Z 1008.697,A -85,B 0,C 180,E1 15110.33,E2 15110.33} C_VEL
LIN {X 0,Y 456.815,Z 1038.263,A -85,B 0,C 180,E1 15111.92,E2 15111.92} C_VEL
LIN {X 0,Y 454.534,Z 1062.901,A -85,B 0,C 180,E1 15114.039,E2 15114.039} C_VEL
LIN {X 0,Y 451.925,Z 1084.665,A -85,B 0,C 180,E1 15116.887,E2 15116.887} C_VEL
LIN {X 0,Y 449.561,Z 1100.282,A -85,B 0,C 180,E1 15120.002,E2 15120.002} C_VEL
LIN {X 0,Y 447.669,Z 1110.554,A -85,B 0,C 180,E1 15123.389,E2 15123.389} C_VEL
LIN {X 0,Y 446.722,Z 1114.463,A -85,B 0,C 180,E1 15125.826,E2 15125.826} C_VEL
LIN {X 0,Y 446.191,Z 1115.706,A -85,B 0,C 180,E1 15127.788,E2 15127.788} C_VEL
LIN {X 0,Y 445.925,Z 1114.576,A -85,B 0,C 180,E1 15130.604,E2 15130.604} C_VEL
LIN {X 0,Y 446.157,Z 1107.302,A -85,B 0,C 180,E1 15134.487,E2 15134.487} C_VEL
LIN {X 0,Y 446.774,Z 1094.423,A -85,B 0,C 180,E1 15137.993,E2 15137.993} C_VEL
LIN {X 0,Y 447.823,Z 1077.121,A -85,B 0,C 180,E1 15141.012,E2 15141.012} C_VEL
LIN {X 0,Y 449.19,Z 1055.311,A -85,B 0,C 180,E1 15143.617,E2 15143.617} C_VEL
LIN {X 0,Y 450.595,Z 1028.285,A -85,B 0,C 180,E1 15145.779,E2 15145.779} C_VEL
LIN {X 0,Y 451.549,Z 998.441,A -85,B 0,C 180,E1 15147.251,E2 15147.251} C_VEL
LIN {X 0,Y 451.42,Z 963.475,A -85,B 0,C 180,E1 15148.118,E2 15148.118} C_VEL
LIN {X 0,Y 442.614,Z 923.03,A -85,B 0,C 180,E1 15149.257,E2 15149.257} C_VEL
LIN {X 0,Y 442.146,Z 923.03,A -85,B 0,C 180,E1 15155.523,E2 15155.523} C_VEL
LIN {X 0,Y 442.036,Z 923.03,A -85,B 0,C 180,E1 15161.21,E2 15161.21} C_VEL
LIN {X 0,Y 442.034,Z 923.03,A -85,B 0,C 180,E1 15166.848,E2 15166.848} C_VEL
LIN {X 0,Y 442.12,Z 923.03,A -85,B 0,C 180,E1 15172.015,E2 15172.015} C_VEL
LIN {X 0,Y 442.256,Z 923.03,A -85,B 0,C 180,E1 15178.675,E2 15178.675} C_VEL
LIN {X 0,Y 442.498,Z 923.03,A -85,B 0,C 180,E1 15183.628,E2 15183.628} C_VEL
LIN {X 0,Y 442.783,Z 923.03,A -85,B 0,C 180,E1 15190.029,E2 15190.029} C_VEL
LIN {X 0,Y 443.038,Z 923.03,A -85,B 0,C 180,E1 15196.171,E2 15196.171} C_VEL
LIN {X 0,Y 443.394,Z 923.03,A -85,B 0,C 180,E1 15202.148,E2 15202.148} C_VEL
LIN {X 0,Y 443.805,Z 923.03,A -85,B 0,C 180,E1 15208.032,E2 15208.032} C_VEL
LIN {X 0,Y 443.64,Z 923.03,A -85,B 0,C 180,E1 15213.889,E2 15213.889} C_VEL
LIN {X 0,Y 443.312,Z 923.03,A -85,B 0,C 180,E1 15219.795,E2 15219.795} C_VEL
LIN {X 0,Y 442.97,Z 923.03,A -85,B 0,C 180,E1 15225.818,E2 15225.818} C_VEL
LIN {X 0,Y 442.657,Z 923.03,A -85,B 0,C 180,E1 15232.035,E2 15232.035} C_VEL
LIN {X 0,Y 442.443,Z 923.03,A -85,B 0,C 180,E1 15238.542,E2 15238.542} C_VEL
LIN {X 0,Y 442.231,Z 923.03,A -85,B 0,C 180,E1 15245.488,E2 15245.488} C_VEL
LIN {X 0,Y 442.107,Z 923.03,A -85,B 0,C 180,E1 15251.237,E2 15251.237} C_VEL
LIN {X 0,Y 442.102,Z 923.03,A -85,B 0,C 180,E1 15256.872,E2 15256.872} C_VEL
LIN {X 0,Y 442.312,Z 923.623,A -85,B 0,C 180,E1 15262.256,E2 15262.256} C_VEL
LIN {X 0,Y 458.08,Z 966.914,A -85,B 0,C 180,E1 15264.694,E2 15264.694} C_VEL
LIN {X 0,Y 468.76,Z 1002.102,A -85,B 0,C 180,E1 15267.08,E2 15267.08} C_VEL
LIN {X 0,Y 463.687,Z 1041.616,A -85,B 0,C 180,E1 15269.571,E2 15269.571} C_VEL
LIN {X 0,Y 458.725,Z 1075.556,A -85,B 0,C 180,E1 15272.535,E2 15272.535} C_VEL
LIN {X 0,Y 454.007,Z 1105.502,A -85,B 0,C 180,E1 15276.028,E2 15276.028} C_VEL
LIN {X 0,Y 449.858,Z 1131.57,A -85,B 0,C 180,E1 15280.077,E2 15280.077} C_VEL
LIN {X 0,Y 446.937,Z 1152.774,A -85,B 0,C 180,E1 15284.556,E2 15284.556} C_VEL
LIN {X 0,Y 445.23,Z 1168.162,A -85,B 0,C 180,E1 15289.158,E2 15289.158} C_VEL
LIN {X 0,Y 444.342,Z 1178.768,A -85,B 0,C 180,E1 15294.142,E2 15294.142} C_VEL
LIN {X 0,Y 444.197,Z 1182.993,A -85,B 0,C 180,E1 15298.048,E2 15298.048} C_VEL
LIN {X 0,Y 444.213,Z 1183.941,A -85,B 0,C 180,E1 15301.947,E2 15301.947} C_VEL
LIN {X 0,Y 444.794,Z 1180.401,A -85,B 0,C 180,E1 15306.827,E2 15306.827} C_VEL
LIN {X 0,Y 446.115,Z 1171.563,A -85,B 0,C 180,E1 15311.724,E2 15311.724} C_VEL
LIN {X 0,Y 448.753,Z 1157.169,A -85,B 0,C 180,E1 15316.565,E2 15316.565} C_VEL
LIN {X 0,Y 453.059,Z 1136.781,A -85,B 0,C 180,E1 15321.271,E2 15321.271} C_VEL
LIN {X 0,Y 459.04,Z 1110.607,A -85,B 0,C 180,E1 15325.596,E2 15325.596} C_VEL
LIN {X 0,Y 466.061,Z 1079.688,A -85,B 0,C 180,E1 15329.364,E2 15329.364} C_VEL
LIN {X 0,Y 473.753,Z 1043.552,A -85,B 0,C 180,E1 15332.603,E2 15332.603} C_VEL
LIN {X 0,Y 480.414,Z 1007.108,A -85,B 0,C 180,E1 15335.028,E2 15335.028} C_VEL
LIN {X 0,Y 477.893,Z 986.285,A -85,B 0,C 180,E1 15337.132,E2 15337.132} C_VEL
LIN {X 0,Y 473.453,Z 971.608,A -85,B 0,C 180,E1 15339.401,E2 15339.401} C_VEL
LIN {X 0,Y 470.044,Z 963.409,A -85,B 0,C 180,E1 15341.552,E2 15341.552} C_VEL
LIN {X 0,Y 469.307,Z 960.405,A -85,B 0,C 180,E1 15342.542,E2 15342.542} C_VEL
LIN {X 0,Y 468.826,Z 959.917,A -85,B 0,C 180,E1 15345.829,E2 15345.829} C_VEL
LIN {X 0,Y 469.779,Z 962.107,A -85,B 0,C 180,E1 15346.962,E2 15346.962} C_VEL
LIN {X 0,Y 473.705,Z 970.093,A -85,B 0,C 180,E1 15349.31,E2 15349.31} C_VEL
LIN {X 0,Y 479.192,Z 985.493,A -85,B 0,C 180,E1 15351.659,E2 15351.659} C_VEL
LIN {X 0,Y 482.87,Z 1003.457,A -85,B 0,C 180,E1 15353.401,E2 15353.401} C_VEL
LIN {X 0,Y 475.056,Z 1047.119,A -85,B 0,C 180,E1 15355.513,E2 15355.513} C_VEL
LIN {X 0,Y 467.006,Z 1087.554,A -85,B 0,C 180,E1 15358.3,E2 15358.3} C_VEL
LIN {X 0,Y 459.836,Z 1123.496,A -85,B 0,C 180,E1 15361.699,E2 15361.699} C_VEL
LIN {X 0,Y 453.66,Z 1154.937,A -85,B 0,C 180,E1 15365.678,E2 15365.678} C_VEL
LIN {X 0,Y 448.947,Z 1180.912,A -85,B 0,C 180,E1 15370.095,E2 15370.095} C_VEL
LIN {X 0,Y 445.967,Z 1201.14,A -85,B 0,C 180,E1 15374.829,E2 15374.829} C_VEL
LIN {X 0,Y 444.582,Z 1215.56,A -85,B 0,C 180,E1 15379.739,E2 15379.739} C_VEL
LIN {X 0,Y 444.199,Z 1223.533,A -85,B 0,C 180,E1 15384.16,E2 15384.16} C_VEL
LIN {X 0,Y 444.156,Z 1226.711,A -85,B 0,C 180,E1 15388.068,E2 15388.068} C_VEL
LIN {X 0,Y 444.206,Z 1226.066,A -85,B 0,C 180,E1 15392.334,E2 15392.334} C_VEL
LIN {X 0,Y 444.291,Z 1221.094,A -85,B 0,C 180,E1 15396.681,E2 15396.681} C_VEL
LIN {X 0,Y 441.887,Z 1217.983,A -85,B 0,C 180,E1 15398.301,E2 15398.301} C_VEL
LIN {X 0,Y 436.826,Z 1212.216,A -85,B 0,C 180,E1 15400.695,E2 15400.695} C_VEL
LIN {X 0,Y 436.783,Z 1211.446,A -85,B 0,C 180,E1 15400.968,E2 15400.968} C_VEL
LIN {X 0,Y 438.166,Z 1195.704,A -85,B 0,C 180,E1 15405.708,E2 15405.708} C_VEL
LIN {X 0,Y 440.947,Z 1173.891,A -85,B 0,C 180,E1 15410.319,E2 15410.319} C_VEL
LIN {X 0,Y 444.875,Z 1148.11,A -85,B 0,C 180,E1 15414.337,E2 15414.337} C_VEL
LIN {X 0,Y 449.731,Z 1117.585,A -85,B 0,C 180,E1 15417.914,E2 15417.914} C_VEL
LIN {X 0,Y 455.229,Z 1082.333,A -85,B 0,C 180,E1 15420.981,E2 15420.981} C_VEL
LIN {X 0,Y 460.689,Z 1042.786,A -85,B 0,C 180,E1 15423.437,E2 15423.437} C_VEL
LIN {X 0,Y 464.329,Z 1002.426,A -85,B 0,C 180,E1 15425.153,E2 15425.153} C_VEL
LIN {X 0,Y 447.691,Z 957.155,A -85,B 0,C 180,E1 15427.516,E2 15427.516} C_VEL
LIN {X 0,Y 434.326,Z 923.03,A -85,B 0,C 180,E1 15429.313,E2 15429.313} C_VEL
LIN {X 0,Y 434.112,Z 923.03,A -85,B 0,C 180,E1 15435.882,E2 15435.882} C_VEL
LIN {X 0,Y 434.126,Z 923.03,A -85,B 0,C 180,E1 15441.207,E2 15441.207} C_VEL
LIN {X 0,Y 434.333,Z 923.03,A -85,B 0,C 180,E1 15448.545,E2 15448.545} C_VEL
LIN {X 0,Y 434.548,Z 923.03,A -85,B 0,C 180,E1 15455.339,E2 15455.339} C_VEL
LIN {X 0,Y 434.736,Z 923.03,A -85,B 0,C 180,E1 15461.772,E2 15461.772} C_VEL
LIN {X 0,Y 434.968,Z 923.286,A -85,B 0,C 180,E1 15465.973,E2 15465.973} C_VEL
LIN {X 0,Y 448.939,Z 957.704,A -85,B 0,C 180,E1 15468.178,E2 15468.178} C_VEL
LIN {X 0,Y 452.518,Z 972.35,A -85,B 0,C 180,E1 15468.831,E2 15468.831} C_VEL
LIN {X 0,Y 451.478,Z 1010.242,A -85,B 0,C 180,E1 15469.903,E2 15469.903} C_VEL
LIN {X 0,Y 449.843,Z 1038.335,A -85,B 0,C 180,E1 15471.429,E2 15471.429} C_VEL
LIN {X 0,Y 447.414,Z 1063.188,A -85,B 0,C 180,E1 15473.579,E2 15473.579} C_VEL
LIN {X 0,Y 444.727,Z 1084.5,A -85,B 0,C 180,E1 15476.349,E2 15476.349} C_VEL
LIN {X 0,Y 442.157,Z 1100.547,A -85,B 0,C 180,E1 15479.513,E2 15479.513} C_VEL
LIN {X 0,Y 440.096,Z 1111.155,A -85,B 0,C 180,E1 15482.954,E2 15482.954} C_VEL
LIN {X 0,Y 438.871,Z 1115.792,A -85,B 0,C 180,E1 15485.931,E2 15485.931} C_VEL
LIN {X 0,Y 438.365,Z 1116.774,A -85,B 0,C 180,E1 15487.928,E2 15487.928} C_VEL
LIN {X 0,Y 438.101,Z 1115.219,A -85,B 0,C 180,E1 15490.796,E2 15490.796} C_VEL
LIN {X 0,Y 438.302,Z 1107.995,A -85,B 0,C 180,E1 15494.552,E2 15494.552} C_VEL
LIN {X 0,Y 438.93,Z 1095.166,A -85,B 0,C 180,E1 15498.052,E2 15498.052} C_VEL
LIN {X 0,Y 440.02,Z 1077.828,A -85,B 0,C 180,E1 15501.108,E2 15501.108} C_VEL
LIN {X 0,Y 441.43,Z 1054.885,A -85,B 0,C 180,E1 15503.854,E2 15503.854} C_VEL
LIN {X 0,Y 442.911,Z 1027.282,A -85,B 0,C 180,E1 15506.047,E2 15506.047} C_VEL
LIN {X 0,Y 443.85,Z 997.415,A -85,B 0,C 180,E1 15507.49,E2 15507.49} C_VEL
LIN {X 0,Y 443.47,Z 963.666,A -85,B 0,C 180,E1 15508.332,E2 15508.332} C_VEL
LIN {X 0,Y 434.666,Z 923.03,A -85,B 0,C 180,E1 15509.536,E2 15509.536} C_VEL
LIN {X 0,Y 434.124,Z 923.03,A -85,B 0,C 180,E1 15516.792,E2 15516.792} C_VEL
LIN {X 0,Y 434.107,Z 923.03,A -85,B 0,C 180,E1 15523.01,E2 15523.01} C_VEL
LIN {X 0,Y 434.138,Z 923.03,A -85,B 0,C 180,E1 15529.977,E2 15529.977} C_VEL
LIN {X 0,Y 434.292,Z 923.03,A -85,B 0,C 180,E1 15536.627,E2 15536.627} C_VEL
LIN {X 0,Y 434.584,Z 923.03,A -85,B 0,C 180,E1 15543.109,E2 15543.109} C_VEL
LIN {X 0,Y 434.832,Z 923.03,A -85,B 0,C 180,E1 15549.771,E2 15549.771} C_VEL
LIN {X 0,Y 435.115,Z 923.03,A -85,B 0,C 180,E1 15556.517,E2 15556.517} C_VEL
LIN {X 0,Y 435.49,Z 923.03,A -85,B 0,C 180,E1 15562.005,E2 15562.005} C_VEL
LIN {X 0,Y 435.922,Z 923.03,A -85,B 0,C 180,E1 15567.996,E2 15567.996} C_VEL
LIN {X 0,Y 435.728,Z 923.03,A -85,B 0,C 180,E1 15573.959,E2 15573.959} C_VEL
LIN {X 0,Y 435.377,Z 923.03,A -85,B 0,C 180,E1 15579.975,E2 15579.975} C_VEL
LIN {X 0,Y 435.051,Z 923.03,A -85,B 0,C 180,E1 15586.113,E2 15586.113} C_VEL
LIN {X 0,Y 434.708,Z 923.03,A -85,B 0,C 180,E1 15592.46,E2 15592.46} C_VEL
LIN {X 0,Y 434.453,Z 923.03,A -85,B 0,C 180,E1 15599.117,E2 15599.117} C_VEL
LIN {X 0,Y 434.341,Z 923.03,A -85,B 0,C 180,E1 15603.8,E2 15603.8} C_VEL
LIN {X 0,Y 434.157,Z 923.03,A -85,B 0,C 180,E1 15610.026,E2 15610.026} C_VEL
LIN {X 0,Y 434.208,Z 923.03,A -85,B 0,C 180,E1 15615.888,E2 15615.888} C_VEL
LIN {X 0,Y 434.321,Z 923.03,A -85,B 0,C 180,E1 15621.675,E2 15621.675} C_VEL
LIN {X 0,Y 449.913,Z 966.362,A -85,B 0,C 180,E1 15624.163,E2 15624.163} C_VEL
LIN {X 0,Y 461.367,Z 1003.88,A -85,B 0,C 180,E1 15626.773,E2 15626.773} C_VEL
LIN {X 0,Y 456.298,Z 1042.163,A -85,B 0,C 180,E1 15629.235,E2 15629.235} C_VEL
LIN {X 0,Y 451.234,Z 1076.012,A -85,B 0,C 180,E1 15632.236,E2 15632.236} C_VEL
LIN {X 0,Y 446.404,Z 1105.839,A -85,B 0,C 180,E1 15635.765,E2 15635.765} C_VEL
LIN {X 0,Y 442.034,Z 1132.663,A -85,B 0,C 180,E1 15640.008,E2 15640.008} C_VEL
LIN {X 0,Y 438.921,Z 1154.612,A -85,B 0,C 180,E1 15644.804,E2 15644.804} C_VEL
LIN {X 0,Y 437.215,Z 1169.904,A -85,B 0,C 180,E1 15649.624,E2 15649.624} C_VEL
LIN {X 0,Y 436.454,Z 1178.967,A -85,B 0,C 180,E1 15654.036,E2 15654.036} C_VEL
LIN {X 0,Y 436.323,Z 1183.335,A -85,B 0,C 180,E1 15658.013,E2 15658.013} C_VEL
LIN {X 0,Y 436.339,Z 1184.385,A -85,B 0,C 180,E1 15661.982,E2 15661.982} C_VEL
LIN {X 0,Y 436.945,Z 1180.988,A -85,B 0,C 180,E1 15666.95,E2 15666.95} C_VEL
LIN {X 0,Y 438.361,Z 1172.304,A -85,B 0,C 180,E1 15671.934,E2 15671.934} C_VEL
LIN {X 0,Y 441.329,Z 1157.512,A -85,B 0,C 180,E1 15677.026,E2 15677.026} C_VEL
LIN {X 0,Y 446.069,Z 1136.726,A -85,B 0,C 180,E1 15681.876,E2 15681.876} C_VEL
LIN {X 0,Y 452.063,Z 1112.171,A -85,B 0,C 180,E1 15686.02,E2 15686.02} C_VEL
LIN {X 0,Y 459.462,Z 1081.786,A -85,B 0,C 180,E1 15689.828,E2 15689.828} C_VEL
LIN {X 0,Y 467.706,Z 1045.978,A -85,B 0,C 180,E1 15693.147,E2 15693.147} C_VEL
LIN {X 0,Y 474.933,Z 1010.024,A -85,B 0,C 180,E1 15695.62,E2 15695.62} C_VEL
LIN {X 0,Y 473.312,Z 991.643,A -85,B 0,C 180,E1 15697.563,E2 15697.563} C_VEL
LIN {X 0,Y 469.951,Z 978.205,A -85,B 0,C 180,E1 15699.708,E2 15699.708} C_VEL
LIN {X 0,Y 467.123,Z 970.075,A -85,B 0,C 180,E1 15701.955,E2 15701.955} C_VEL
LIN {X 0,Y 466.57,Z 967.768,A -85,B 0,C 180,E1 15702.851,E2 15702.851} C_VEL
LIN {X 0,Y 466.26,Z 967.326,A -85,B 0,C 180,E1 15705.476,E2 15705.476} C_VEL
LIN {X 0,Y 467.862,Z 971.306,A -85,B 0,C 180,E1 15707.434,E2 15707.434} C_VEL
LIN {X 0,Y 471.497,Z 979.895,A -85,B 0,C 180,E1 15709.58,E2 15709.58} C_VEL
LIN {X 0,Y 475.773,Z 994.965,A -85,B 0,C 180,E1 15711.694,E2 15711.694} C_VEL
LIN {X 0,Y 477.237,Z 1007.201,A -85,B 0,C 180,E1 15712.815,E2 15712.815} C_VEL
LIN {X 0,Y 468.723,Z 1050.326,A -85,B 0,C 180,E1 15715.024,E2 15715.024} C_VEL
LIN {X 0,Y 460.167,Z 1090.344,A -85,B 0,C 180,E1 15717.912,E2 15717.912} C_VEL
LIN {X 0,Y 452.229,Z 1127.408,A -85,B 0,C 180,E1 15721.587,E2 15721.587} C_VEL
LIN {X 0,Y 445.735,Z 1158.393,A -85,B 0,C 180,E1 15725.75,E2 15725.75} C_VEL
LIN {X 0,Y 440.912,Z 1183.456,A -85,B 0,C 180,E1 15730.276,E2 15730.276} C_VEL
LIN {X 0,Y 438.042,Z 1202.457,A -85,B 0,C 180,E1 15734.987,E2 15734.987} C_VEL
LIN {X 0,Y 436.702,Z 1215.3,A -85,B 0,C 180,E1 15739.552,E2 15739.552} C_VEL
LIN {X 0,Y 436.302,Z 1223.218,A -85,B 0,C 180,E1 15744.054,E2 15744.054} C_VEL
LIN {X 0,Y 436.27,Z 1226.306,A -85,B 0,C 180,E1 15748.033,E2 15748.033} C_VEL
LIN {X 0,Y 436.361,Z 1225.878,A -85,B 0,C 180,E1 15752.002,E2 15752.002} C_VEL
LIN {X 0,Y 436.438,Z 1220.213,A -85,B 0,C 180,E1 15756.977,E2 15756.977} C_VEL
LIN {X 0,Y 436.783,Z 1211.446,A -85,B 0,C 180,E1 15760.968,E2 15760.968} C_VEL
LIN {X 0,Y 434.63,Z 1206.811,A -85,B 0,C 180,E1 15762.558,E2 15762.558} C_VEL
LIN {X 0,Y 430.033,Z 1198.885,A -85,B 0,C 180,E1 15764.897,E2 15764.897} C_VEL
LIN {X 0,Y 430.033,Z 1197.921,A -85,B 0,C 180,E1 15765.162,E2 15765.162} C_VEL
LIN {X 0,Y 432.596,Z 1177.413,A -85,B 0,C 180,E1 15769.802,E2 15769.802} C_VEL
LIN {X 0,Y 436.855,Z 1150.193,A -85,B 0,C 180,E1 15774.271,E2 15774.271} C_VEL
LIN {X 0,Y 441.973,Z 1118.705,A -85,B 0,C 180,E1 15778.086,E2 15778.086} C_VEL
LIN {X 0,Y 447.48,Z 1084.525,A -85,B 0,C 180,E1 15781.154,E2 15781.154} C_VEL
LIN {X 0,Y 452.933,Z 1046.057,A -85,B 0,C 180,E1 15783.654,E2 15783.654} C_VEL
LIN {X 0,Y 457.107,Z 1004.472,A -85,B 0,C 180,E1 15785.5,E2 15785.5} C_VEL
LIN {X 0,Y 440.991,Z 960.276,A -85,B 0,C 180,E1 15787.883,E2 15787.883} C_VEL
LIN {X 0,Y 426.334,Z 923.03,A -85,B 0,C 180,E1 15789.97,E2 15789.97} C_VEL
LIN {X 0,Y 426.194,Z 923.03,A -85,B 0,C 180,E1 15795.183,E2 15795.183} C_VEL
LIN {X 0,Y 426.234,Z 923.03,A -85,B 0,C 180,E1 15801.278,E2 15801.278} C_VEL
LIN {X 0,Y 426.418,Z 923.03,A -85,B 0,C 180,E1 15808.29,E2 15808.29} C_VEL
LIN {X 0,Y 426.643,Z 923.03,A -85,B 0,C 180,E1 15814.85,E2 15814.85} C_VEL
LIN {X 0,Y 426.815,Z 923.03,A -85,B 0,C 180,E1 15821.422,E2 15821.422} C_VEL
LIN {X 0,Y 426.97,Z 923.03,A -85,B 0,C 180,E1 15825.135,E2 15825.135} C_VEL
LIN {X 0,Y 441.87,Z 958.68,A -85,B 0,C 180,E1 15827.625,E2 15827.625} C_VEL
LIN {X 0,Y 445.715,Z 974.394,A -85,B 0,C 180,E1 15828.357,E2 15828.357} C_VEL
LIN {X 0,Y 444.549,Z 1011.442,A -85,B 0,C 180,E1 15829.442,E2 15829.442} C_VEL
LIN {X 0,Y 442.74,Z 1040.183,A -85,B 0,C 180,E1 15831.044,E2 15831.044} C_VEL
LIN {X 0,Y 440.178,Z 1064.815,A -85,B 0,C 180,E1 15833.225,E2 15833.225} C_VEL
LIN {X 0,Y 437.327,Z 1085.848,A -85,B 0,C 180,E1 15836.039,E2 15836.039} C_VEL
LIN {X 0,Y 434.793,Z 1100.809,A -85,B 0,C 180,E1 15839.006,E2 15839.006} C_VEL
LIN {X 0,Y 432.528,Z 1111.73,A -85,B 0,C 180,E1 15842.482,E2 15842.482} C_VEL
LIN {X 0,Y 431.038,Z 1117.076,A -85,B 0,C 180,E1 15846.039,E2 15846.039} C_VEL
LIN {X 0,Y 430.504,Z 1117.76,A -85,B 0,C 180,E1 15848.073,E2 15848.073} C_VEL
LIN {X 0,Y 430.267,Z 1115.664,A -85,B 0,C 180,E1 15851.157,E2 15851.157} C_VEL
LIN {X 0,Y 430.483,Z 1108.042,A -85,B 0,C 180,E1 15854.823,E2 15854.823} C_VEL
LIN {X 0,Y 431.178,Z 1094.635,A -85,B 0,C 180,E1 15858.388,E2 15858.388} C_VEL
LIN {X 0,Y 432.329,Z 1076.984,A -85,B 0,C 180,E1 15861.437,E2 15861.437} C_VEL
LIN {X 0,Y 433.727,Z 1053.751,A -85,B 0,C 180,E1 15864.167,E2 15864.167} C_VEL
LIN {X 0,Y 435.197,Z 1026.941,A -85,B 0,C 180,E1 15866.274,E2 15866.274} C_VEL
LIN {X 0,Y 436.15,Z 996.064,A -85,B 0,C 180,E1 15867.748,E2 15867.748} C_VEL
LIN {X 0,Y 435.617,Z 964.033,A -85,B 0,C 180,E1 15868.541,E2 15868.541} C_VEL
LIN {X 0,Y 426.718,Z 923.03,A -85,B 0,C 180,E1 15869.723,E2 15869.723} C_VEL
LIN {X 0,Y 426.193,Z 923.03,A -85,B 0,C 180,E1 15877.07,E2 15877.07} C_VEL
LIN {X 0,Y 426.186,Z 923.03,A -85,B 0,C 180,E1 15882.354,E2 15882.354} C_VEL
LIN {X 0,Y 426.215,Z 923.03,A -85,B 0,C 180,E1 15888.122,E2 15888.122} C_VEL
LIN {X 0,Y 426.208,Z 923.03,A -85,B 0,C 180,E1 15894.636,E2 15894.636} C_VEL
LIN {X 0,Y 426.496,Z 923.03,A -85,B 0,C 180,E1 15900.245,E2 15900.245} C_VEL
LIN {X 0,Y 426.762,Z 923.03,A -85,B 0,C 180,E1 15907.06,E2 15907.06} C_VEL
LIN {X 0,Y 427.051,Z 923.03,A -85,B 0,C 180,E1 15913.539,E2 15913.539} C_VEL
LIN {X 0,Y 427.411,Z 923.03,A -85,B 0,C 180,E1 15919.801,E2 15919.801} C_VEL
LIN {X 0,Y 427.907,Z 923.03,A -85,B 0,C 180,E1 15925.932,E2 15925.932} C_VEL
LIN {X 0,Y 428.025,Z 923.03,A -85,B 0,C 180,E1 15932.005,E2 15932.005} C_VEL
LIN {X 0,Y 427.556,Z 923.03,A -85,B 0,C 180,E1 15938.258,E2 15938.258} C_VEL
LIN {X 0,Y 427.237,Z 923.03,A -85,B 0,C 180,E1 15944.315,E2 15944.315} C_VEL
LIN {X 0,Y 426.866,Z 923.03,A -85,B 0,C 180,E1 15950.711,E2 15950.711} C_VEL
LIN {X 0,Y 426.573,Z 923.03,A -85,B 0,C 180,E1 15957.67,E2 15957.67} C_VEL
LIN {X 0,Y 426.322,Z 923.03,A -85,B 0,C 180,E1 15964.524,E2 15964.524} C_VEL
LIN {X 0,Y 426.271,Z 923.03,A -85,B 0,C 180,E1 15969.622,E2 15969.622} C_VEL
LIN {X 0,Y 426.257,Z 923.03,A -85,B 0,C 180,E1 15975.123,E2 15975.123} C_VEL
LIN {X 0,Y 426.349,Z 923.638,A -85,B 0,C 180,E1 15981.142,E2 15981.142} C_VEL
LIN {X 0,Y 442.289,Z 967.168,A -85,B 0,C 180,E1 15983.713,E2 15983.713} C_VEL
LIN {X 0,Y 453.617,Z 1004.281,A -85,B 0,C 180,E1 15986.35,E2 15986.35} C_VEL
LIN {X 0,Y 449.164,Z 1041.251,A -85,B 0,C 180,E1 15988.778,E2 15988.778} C_VEL
LIN {X 0,Y 443.867,Z 1075.45,A -85,B 0,C 180,E1 15991.825,E2 15991.825} C_VEL
LIN {X 0,Y 438.985,Z 1104.922,A -85,B 0,C 180,E1 15995.329,E2 15995.329} C_VEL
LIN {X 0,Y 434.667,Z 1130.697,A -85,B 0,C 180,E1 15999.389,E2 15999.389} C_VEL
LIN {X 0,Y 431.607,Z 1151.23,A -85,B 0,C 180,E1 16003.732,E2 16003.732} C_VEL
LIN {X 0,Y 429.658,Z 1166.93,A -85,B 0,C 180,E1 16008.331,E2 16008.331} C_VEL
LIN {X 0,Y 428.684,Z 1177.442,A -85,B 0,C 180,E1 16012.918,E2 16012.918} C_VEL
LIN {X 0,Y 428.427,Z 1183.675,A -85,B 0,C 180,E1 16017.977,E2 16017.977} C_VEL
LIN {X 0,Y 428.451,Z 1184.834,A -85,B 0,C 180,E1 16022.019,E2 16022.019} C_VEL
LIN {X 0,Y 429.123,Z 1181.589,A -85,B 0,C 180,E1 16027.077,E2 16027.077} C_VEL
LIN {X 0,Y 430.63,Z 1173.073,A -85,B 0,C 180,E1 16032.152,E2 16032.152} C_VEL
LIN {X 0,Y 433.697,Z 1158.835,A -85,B 0,C 180,E1 16037.225,E2 16037.225} C_VEL
LIN {X 0,Y 438.848,Z 1138.022,A -85,B 0,C 180,E1 16042.255,E2 16042.255} C_VEL
LIN {X 0,Y 445.58,Z 1112.179,A -85,B 0,C 180,E1 16046.699,E2 16046.699} C_VEL
LIN {X 0,Y 453.464,Z 1081.927,A -85,B 0,C 180,E1 16050.54,E2 16050.54} C_VEL
LIN {X 0,Y 462.629,Z 1044.717,A -85,B 0,C 180,E1 16054.009,E2 16054.009} C_VEL
LIN {X 0,Y 469.662,Z 1011.201,A -85,B 0,C 180,E1 16056.405,E2 16056.405} C_VEL
LIN {X 0,Y 468.385,Z 994.356,A -85,B 0,C 180,E1 16058.37,E2 16058.37} C_VEL
LIN {X 0,Y 465.685,Z 982.077,A -85,B 0,C 180,E1 16060.652,E2 16060.652} C_VEL
LIN {X 0,Y 463.822,Z 975.088,A -85,B 0,C 180,E1 16063.167,E2 16063.167} C_VEL
LIN {X 0,Y 463.979,Z 975.214,A -85,B 0,C 180,E1 16065.763,E2 16065.763} C_VEL
LIN {X 0,Y 466.272,Z 981.679,A -85,B 0,C 180,E1 16068.189,E2 16068.189} C_VEL
LIN {X 0,Y 469.768,Z 993.144,A -85,B 0,C 180,E1 16070.344,E2 16070.344} C_VEL
LIN {X 0,Y 472.146,Z 1008.901,A -85,B 0,C 180,E1 16072.116,E2 16072.116} C_VEL
LIN {X 0,Y 462.923,Z 1051.682,A -85,B 0,C 180,E1 16074.391,E2 16074.391} C_VEL
LIN {X 0,Y 453.909,Z 1090.626,A -85,B 0,C 180,E1 16077.273,E2 16077.273} C_VEL
LIN {X 0,Y 445.293,Z 1128.152,A -85,B 0,C 180,E1 16081.104,E2 16081.104} C_VEL
LIN {X 0,Y 438.438,Z 1158.707,A -85,B 0,C 180,E1 16085.32,E2 16085.32} C_VEL
LIN {X 0,Y 433.398,Z 1183.33,A -85,B 0,C 180,E1 16089.88,E2 16089.88} C_VEL
LIN {X 0,Y 430.262,Z 1202.338,A -85,B 0,C 180,E1 16094.709,E2 16094.709} C_VEL
LIN {X 0,Y 428.774,Z 1216.167,A -85,B 0,C 180,E1 16099.87,E2 16099.87} C_VEL
LIN {X 0,Y 428.405,Z 1222.889,A -85,B 0,C 180,E1 16103.944,E2 16103.944} C_VEL
LIN {X 0,Y 428.374,Z 1225.904,A -85,B 0,C 180,E1 16107.996,E2 16107.996} C_VEL
LIN {X 0,Y 428.466,Z 1225.402,A -85,B 0,C 180,E1 16112.039,E2 16112.039} C_VEL
LIN {X 0,Y 428.548,Z 1219.592,A -85,B 0,C 180,E1 16117.106,E2 16117.106} C_VEL
LIN {X 0,Y 429.093,Z 1209.19,A -85,B 0,C 180,E1 16121.7,E2 16121.7} C_VEL
LIN {X 0,Y 430.033,Z 1197.921,A -85,B 0,C 180,E1 16125.162,E2 16125.162} C_VEL
LIN {X 0,Y 427.019,Z 1189.935,A -85,B 0,C 180,E1 16127.211,E2 16127.211} C_VEL
LIN {X 0,Y 424.294,Z 1180.912,A -85,B 0,C 180,E1 16129.21,E2 16129.21} C_VEL
LIN {X 0,Y 428.195,Z 1155.865,A -85,B 0,C 180,E1 16133.641,E2 16133.641} C_VEL
LIN {X 0,Y 433.143,Z 1126.194,A -85,B 0,C 180,E1 16137.549,E2 16137.549} C_VEL
LIN {X 0,Y 439.041,Z 1091.017,A -85,B 0,C 180,E1 16140.98,E2 16140.98} C_VEL
LIN {X 0,Y 444.787,Z 1052.193,A -85,B 0,C 180,E1 16143.691,E2 16143.691} C_VEL
LIN {X 0,Y 449.713,Z 1011.418,A -85,B 0,C 180,E1 16145.637,E2 16145.637} C_VEL
LIN {X 0,Y 449.212,Z 1004.561,A -85,B 0,C 180,E1 16145.963,E2 16145.963} C_VEL
LIN {X 0,Y 432.754,Z 959.752,A -85,B 0,C 180,E1 16148.454,E2 16148.454} C_VEL
LIN {X 0,Y 418.373,Z 923.03,A -85,B 0,C 180,E1 16150.571,E2 16150.571} C_VEL
LIN {X 0,Y 418.194,Z 923.03,A -85,B 0,C 180,E1 16156.646,E2 16156.646} C_VEL
LIN {X 0,Y 418.321,Z 923.03,A -85,B 0,C 180,E1 16162.65,E2 16162.65} C_VEL
LIN {X 0,Y 418.544,Z 923.03,A -85,B 0,C 180,E1 16170.08,E2 16170.08} C_VEL
LIN {X 0,Y 418.722,Z 923.03,A -85,B 0,C 180,E1 16176.613,E2 16176.613} C_VEL
LIN {X 0,Y 419.027,Z 923.03,A -85,B 0,C 180,E1 16183.773,E2 16183.773} C_VEL
LIN {X 0,Y 419.029,Z 923.03,A -85,B 0,C 180,E1 16184.242,E2 16184.242} C_VEL
LIN {X 0,Y 434.111,Z 957.591,A -85,B 0,C 180,E1 16186.908,E2 16186.908} C_VEL
LIN {X 0,Y 438.97,Z 974.809,A -85,B 0,C 180,E1 16187.822,E2 16187.822} C_VEL
LIN {X 0,Y 437.753,Z 1012.193,A -85,B 0,C 180,E1 16188.932,E2 16188.932} C_VEL
LIN {X 0,Y 435.86,Z 1040.461,A -85,B 0,C 180,E1 16190.524,E2 16190.524} C_VEL
LIN {X 0,Y 432.988,Z 1066.427,A -85,B 0,C 180,E1 16192.86,E2 16192.86} C_VEL
LIN {X 0,Y 429.967,Z 1087.322,A -85,B 0,C 180,E1 16195.719,E2 16195.719} C_VEL
LIN {X 0,Y 427.093,Z 1103.097,A -85,B 0,C 180,E1 16198.989,E2 16198.989} C_VEL
LIN {X 0,Y 424.969,Z 1112.388,A -85,B 0,C 180,E1 16202.04,E2 16202.04} C_VEL
LIN {X 0,Y 423.556,Z 1117.462,A -85,B 0,C 180,E1 16205.119,E2 16205.119} C_VEL
LIN {X 0,Y 422.639,Z 1118.747,A -85,B 0,C 180,E1 16208.225,E2 16208.225} C_VEL
LIN {X 0,Y 422.407,Z 1116.218,A -85,B 0,C 180,E1 16211.349,E2 16211.349} C_VEL
LIN {X 0,Y 422.718,Z 1107.467,A -85,B 0,C 180,E1 16215.298,E2 16215.298} C_VEL
LIN {X 0,Y 423.4,Z 1093.933,A -85,B 0,C 180,E1 16218.738,E2 16218.738} C_VEL
LIN {X 0,Y 424.686,Z 1074.525,A -85,B 0,C 180,E1 16221.975,E2 16221.975} C_VEL
LIN {X 0,Y 426.129,Z 1051.065,A -85,B 0,C 180,E1 16224.627,E2 16224.627} C_VEL
LIN {X 0,Y 427.62,Z 1023.326,A -85,B 0,C 180,E1 16226.711,E2 16226.711} C_VEL
LIN {X 0,Y 428.484,Z 993.061,A -85,B 0,C 180,E1 16228.058,E2 16228.058} C_VEL
LIN {X 0,Y 427.854,Z 964.969,A -85,B 0,C 180,E1 16228.743,E2 16228.743} C_VEL
LIN {X 0,Y 418.752,Z 923.03,A -85,B 0,C 180,E1 16229.969,E2 16229.969} C_VEL
LIN {X 0,Y 418.285,Z 923.03,A -85,B 0,C 180,E1 16237.892,E2 16237.892} C_VEL
LIN {X 0,Y 418.188,Z 923.03,A -85,B 0,C 180,E1 16243.702,E2 16243.702} C_VEL
LIN {X 0,Y 418.259,Z 923.03,A -85,B 0,C 180,E1 16249.416,E2 16249.416} C_VEL
LIN {X 0,Y 418.324,Z 923.03,A -85,B 0,C 180,E1 16256.187,E2 16256.187} C_VEL
LIN {X 0,Y 418.63,Z 923.03,A -85,B 0,C 180,E1 16261.997,E2 16261.997} C_VEL
LIN {X 0,Y 418.889,Z 923.03,A -85,B 0,C 180,E1 16268.837,E2 16268.837} C_VEL
LIN {X 0,Y 419.231,Z 923.03,A -85,B 0,C 180,E1 16275.368,E2 16275.368} C_VEL
LIN {X 0,Y 419.659,Z 923.03,A -85,B 0,C 180,E1 16281.701,E2 16281.701} C_VEL
LIN {X 0,Y 420.12,Z 923.03,A -85,B 0,C 180,E1 16287.921,E2 16287.921} C_VEL
LIN {X 0,Y 419.905,Z 923.03,A -85,B 0,C 180,E1 16294.109,E2 16294.109} C_VEL
LIN {X 0,Y 419.508,Z 923.03,A -85,B 0,C 180,E1 16300.356,E2 16300.356} C_VEL
LIN {X 0,Y 419.181,Z 923.03,A -85,B 0,C 180,E1 16306.741,E2 16306.741} C_VEL
LIN {X 0,Y 418.797,Z 923.03,A -85,B 0,C 180,E1 16313.362,E2 16313.362} C_VEL
LIN {X 0,Y 418.565,Z 923.03,A -85,B 0,C 180,E1 16320.335,E2 16320.335} C_VEL
LIN {X 0,Y 418.368,Z 923.03,A -85,B 0,C 180,E1 16327.378,E2 16327.378} C_VEL
LIN {X 0,Y 418.269,Z 923.03,A -85,B 0,C 180,E1 16333.732,E2 16333.732} C_VEL
LIN {X 0,Y 418.413,Z 923.651,A -85,B 0,C 180,E1 16340.566,E2 16340.566} C_VEL
LIN {X 0,Y 434.14,Z 966.408,A -85,B 0,C 180,E1 16343.147,E2 16343.147} C_VEL
LIN {X 0,Y 445.854,Z 1004.863,A -85,B 0,C 180,E1 16345.934,E2 16345.934} C_VEL
LIN {X 0,Y 445.277,Z 1017.41,A -85,B 0,C 180,E1 16346.733,E2 16346.733} C_VEL
LIN {X 0,Y 439.956,Z 1053.824,A -85,B 0,C 180,E1 16349.416,E2 16349.416} C_VEL
LIN {X 0,Y 434.5,Z 1086.822,A -85,B 0,C 180,E1 16352.72,E2 16352.72} C_VEL
LIN {X 0,Y 429.418,Z 1116.398,A -85,B 0,C 180,E1 16356.693,E2 16356.693} C_VEL
LIN {X 0,Y 425.284,Z 1141.961,A -85,B 0,C 180,E1 16361.348,E2 16361.348} C_VEL
LIN {X 0,Y 422.559,Z 1160.53,A -85,B 0,C 180,E1 16366.029,E2 16366.029} C_VEL
LIN {X 0,Y 421.185,Z 1174.092,A -85,B 0,C 180,E1 16371.003,E2 16371.003} C_VEL
LIN {X 0,Y 420.56,Z 1182.126,A -85,B 0,C 180,E1 16375.877,E2 16375.877} C_VEL
LIN {X 0,Y 420.42,Z 1185.063,A -85,B 0,C 180,E1 16379.998,E2 16379.998} C_VEL
LIN {X 0,Y 420.719,Z 1184.7,A -85,B 0,C 180,E1 16384.117,E2 16384.117} C_VEL
LIN {X 0,Y 421.769,Z 1179.586,A -85,B 0,C 180,E1 16389.242,E2 16389.242} C_VEL
LIN {X 0,Y 423.936,Z 1169.005,A -85,B 0,C 180,E1 16394.446,E2 16394.446} C_VEL
LIN {X 0,Y 428.072,Z 1152.542,A -85,B 0,C 180,E1 16399.592,E2 16399.592} C_VEL
LIN {X 0,Y 434.141,Z 1130.353,A -85,B 0,C 180,E1 16404.412,E2 16404.412} C_VEL
LIN {X 0,Y 441.635,Z 1103.783,A -85,B 0,C 180,E1 16408.619,E2 16408.619} C_VEL
LIN {X 0,Y 450.33,Z 1072.315,A -85,B 0,C 180,E1 16412.327,E2 16412.327} C_VEL
LIN {X 0,Y 460.288,Z 1033.951,A -85,B 0,C 180,E1 16415.64,E2 16415.64} C_VEL
LIN {X 0,Y 464.578,Z 1015.356,A -85,B 0,C 180,E1 16416.948,E2 16416.948} C_VEL
LIN {X 0,Y 464.019,Z 999.514,A -85,B 0,C 180,E1 16418.874,E2 16418.874} C_VEL
LIN {X 0,Y 462.034,Z 987.677,A -85,B 0,C 180,E1 16421.248,E2 16421.248} C_VEL
LIN {X 0,Y 460.984,Z 982.383,A -85,B 0,C 180,E1 16423.499,E2 16423.499} C_VEL
LIN {X 0,Y 461.494,Z 983.279,A -85,B 0,C 180,E1 16426.081,E2 16426.081} C_VEL
LIN {X 0,Y 463.474,Z 989.61,A -85,B 0,C 180,E1 16428.215,E2 16428.215} C_VEL
LIN {X 0,Y 466.281,Z 1003.106,A -85,B 0,C 180,E1 16430.484,E2 16430.484} C_VEL
LIN {X 0,Y 466.746,Z 1013.086,A -85,B 0,C 180,E1 16431.501,E2 16431.501} C_VEL
LIN {X 0,Y 456.414,Z 1056.813,A -85,B 0,C 180,E1 16433.962,E2 16433.962} C_VEL
LIN {X 0,Y 446.277,Z 1097.532,A -85,B 0,C 180,E1 16437.22,E2 16437.22} C_VEL
LIN {X 0,Y 437.45,Z 1133.031,A -85,B 0,C 180,E1 16441.102,E2 16441.102} C_VEL
LIN {X 0,Y 430.456,Z 1162.585,A -85,B 0,C 180,E1 16445.447,E2 16445.447} C_VEL
LIN {X 0,Y 425.183,Z 1186.859,A -85,B 0,C 180,E1 16450.28,E2 16450.28} C_VEL
LIN {X 0,Y 422.041,Z 1205.591,A -85,B 0,C 180,E1 16455.505,E2 16455.505} C_VEL
LIN {X 0,Y 420.75,Z 1217.724,A -85,B 0,C 180,E1 16460.604,E2 16460.604} C_VEL
LIN {X 0,Y 420.479,Z 1224.466,A -85,B 0,C 180,E1 16465.897,E2 16465.897} C_VEL
LIN {X 0,Y 420.568,Z 1225.655,A -85,B 0,C 180,E1 16470.018,E2 16470.018} C_VEL
LIN {X 0,Y 420.542,Z 1223.243,A -85,B 0,C 180,E1 16474.139,E2 16474.139} C_VEL
LIN {X 0,Y 420.831,Z 1215.834,A -85,B 0,C 180,E1 16478.879,E2 16478.879} C_VEL
LIN {X 0,Y 421.759,Z 1202.03,A -85,B 0,C 180,E1 16484.013,E2 16484.013} C_VEL
LIN {X 0,Y 424.165,Z 1182.131,A -85,B 0,C 180,E1 16488.961,E2 16488.961} C_VEL
LIN {X 0,Y 424.294,Z 1180.912,A -85,B 0,C 180,E1 16489.21,E2 16489.21} C_VEL
LIN {X 0,Y 421.763,Z 1171.239,A -85,B 0,C 180,E1 16491.158,E2 16491.158} C_VEL
LIN {X 0,Y 419.617,Z 1160.78,A -85,B 0,C 180,E1 16493.065,E2 16493.065} C_VEL
LIN {X 0,Y 424.762,Z 1130.838,A -85,B 0,C 180,E1 16497.279,E2 16497.279} C_VEL
LIN {X 0,Y 430.582,Z 1096.895,A -85,B 0,C 180,E1 16500.801,E2 16500.801} C_VEL
LIN {X 0,Y 436.213,Z 1061.083,A -85,B 0,C 180,E1 16503.528,E2 16503.528} C_VEL
LIN {X 0,Y 441.598,Z 1020.3,A -85,B 0,C 180,E1 16505.704,E2 16505.704} C_VEL
LIN {X 0,Y 442.346,Z 1007.734,A -85,B 0,C 180,E1 16506.243,E2 16506.243} C_VEL
LIN {X 0,Y 426.425,Z 963.794,A -85,B 0,C 180,E1 16508.779,E2 16508.779} C_VEL
LIN {X 0,Y 410.367,Z 923.03,A -85,B 0,C 180,E1 16511.132,E2 16511.132} C_VEL
LIN {X 0,Y 410.244,Z 923.03,A -85,B 0,C 180,E1 16518.473,E2 16518.473} C_VEL
LIN {X 0,Y 410.386,Z 923.03,A -85,B 0,C 180,E1 16524.127,E2 16524.127} C_VEL
LIN {X 0,Y 410.63,Z 923.03,A -85,B 0,C 180,E1 16531.422,E2 16531.422} C_VEL
LIN {X 0,Y 410.839,Z 923.03,A -85,B 0,C 180,E1 16538.422,E2 16538.422} C_VEL
LIN {X 0,Y 411.138,Z 923.54,A -85,B 0,C 180,E1 16543.31,E2 16543.31} C_VEL
LIN {X 0,Y 426.524,Z 957.096,A -85,B 0,C 180,E1 16546.177,E2 16546.177} C_VEL
LIN {X 0,Y 432.293,Z 976.059,A -85,B 0,C 180,E1 16547.275,E2 16547.275} C_VEL
LIN {X 0,Y 430.975,Z 1013.586,A -85,B 0,C 180,E1 16548.435,E2 16548.435} C_VEL
LIN {X 0,Y 428.861,Z 1042.619,A -85,B 0,C 180,E1 16550.111,E2 16550.111} C_VEL
LIN {X 0,Y 425.804,Z 1068.14,A -85,B 0,C 180,E1 16552.483,E2 16552.483} C_VEL
LIN {X 0,Y 422.609,Z 1088.826,A -85,B 0,C 180,E1 16555.388,E2 16555.388} C_VEL
LIN {X 0,Y 419.768,Z 1103.466,A -85,B 0,C 180,E1 16558.455,E2 16558.455} C_VEL
LIN {X 0,Y 417.168,Z 1114.168,A -85,B 0,C 180,E1 16562.078,E2 16562.078} C_VEL
LIN {X 0,Y 416.144,Z 1117.687,A -85,B 0,C 180,E1 16564.167,E2 16564.167} C_VEL
LIN {X 0,Y 415.316,Z 1119.538,A -85,B 0,C 180,E1 16566.269,E2 16566.269} C_VEL
LIN {X 0,Y 414.605,Z 1118.499,A -85,B 0,C 180,E1 16570.17,E2 16570.17} C_VEL
LIN {X 0,Y 414.694,Z 1111.248,A -85,B 0,C 180,E1 16574.241,E2 16574.241} C_VEL
LIN {X 0,Y 415.332,Z 1098.452,A -85,B 0,C 180,E1 16577.967,E2 16577.967} C_VEL
LIN {X 0,Y 416.552,Z 1079.583,A -85,B 0,C 180,E1 16581.446,E2 16581.446} C_VEL
LIN {X 0,Y 418.125,Z 1055.715,A -85,B 0,C 180,E1 16584.372,E2 16584.372} C_VEL
LIN {X 0,Y 419.652,Z 1028.201,A -85,B 0,C 180,E1 16586.608,E2 16586.608} C_VEL
LIN {X 0,Y 420.653,Z 998.08,A -85,B 0,C 180,E1 16588.102,E2 16588.102} C_VEL
LIN {X 0,Y 420.38,Z 967.183,A -85,B 0,C 180,E1 16588.906,E2 16588.906} C_VEL
LIN {X 0,Y 410.814,Z 923.03,A -85,B 0,C 180,E1 16590.227,E2 16590.227} C_VEL
LIN {X 0,Y 410.36,Z 923.03,A -85,B 0,C 180,E1 16596.102,E2 16596.102} C_VEL
LIN {X 0,Y 410.233,Z 923.03,A -85,B 0,C 180,E1 16602.527,E2 16602.527} C_VEL
LIN {X 0,Y 410.255,Z 923.03,A -85,B 0,C 180,E1 16608.451,E2 16608.451} C_VEL
LIN {X 0,Y 410.37,Z 923.03,A -85,B 0,C 180,E1 16614.11,E2 16614.11} C_VEL
LIN {X 0,Y 410.675,Z 923.03,A -85,B 0,C 180,E1 16621.405,E2 16621.405} C_VEL
LIN {X 0,Y 410.923,Z 923.03,A -85,B 0,C 180,E1 16628.406,E2 16628.406} C_VEL
LIN {X 0,Y 411.283,Z 923.03,A -85,B 0,C 180,E1 16635.079,E2 16635.079} C_VEL
LIN {X 0,Y 411.735,Z 923.03,A -85,B 0,C 180,E1 16642.289,E2 16642.289} C_VEL
LIN {X 0,Y 412.211,Z 923.03,A -85,B 0,C 180,E1 16647.881,E2 16647.881} C_VEL
LIN {X 0,Y 412.213,Z 923.03,A -85,B 0,C 180,E1 16652.082,E2 16652.082} C_VEL
LIN {X 0,Y 411.756,Z 923.03,A -85,B 0,C 180,E1 16658.422,E2 16658.422} C_VEL
LIN {X 0,Y 411.347,Z 923.03,A -85,B 0,C 180,E1 16664.88,E2 16664.88} C_VEL
LIN {X 0,Y 410.951,Z 923.03,A -85,B 0,C 180,E1 16671.552,E2 16671.552} C_VEL
LIN {X 0,Y 410.69,Z 923.03,A -85,B 0,C 180,E1 16678.552,E2 16678.552} C_VEL
LIN {X 0,Y 410.419,Z 923.03,A -85,B 0,C 180,E1 16685.9,E2 16685.9} C_VEL
LIN {X 0,Y 410.309,Z 923.03,A -85,B 0,C 180,E1 16692.557,E2 16692.557} C_VEL
LIN {X 0,Y 410.459,Z 923.321,A -85,B 0,C 180,E1 16699.968,E2 16699.968} C_VEL
LIN {X 0,Y 426.331,Z 966.808,A -85,B 0,C 180,E1 16702.647,E2 16702.647} C_VEL
LIN {X 0,Y 438.404,Z 1006.425,A -85,B 0,C 180,E1 16705.591,E2 16705.591} C_VEL
LIN {X 0,Y 438.493,Z 1014.421,A -85,B 0,C 180,E1 16706.123,E2 16706.123} C_VEL
LIN {X 0,Y 432.859,Z 1052.338,A -85,B 0,C 180,E1 16708.897,E2 16708.897} C_VEL
LIN {X 0,Y 427.357,Z 1085.217,A -85,B 0,C 180,E1 16712.185,E2 16712.185} C_VEL
LIN {X 0,Y 422.081,Z 1114.912,A -85,B 0,C 180,E1 16716.163,E2 16716.163} C_VEL
LIN {X 0,Y 417.841,Z 1139.983,A -85,B 0,C 180,E1 16720.686,E2 16720.686} C_VEL
LIN {X 0,Y 414.792,Z 1160.343,A -85,B 0,C 180,E1 16725.762,E2 16725.762} C_VEL
LIN {X 0,Y 413.325,Z 1174.264,A -85,B 0,C 180,E1 16730.885,E2 16730.885} C_VEL
LIN {X 0,Y 412.668,Z 1182.342,A -85,B 0,C 180,E1 16735.798,E2 16735.798} C_VEL
LIN {X 0,Y 412.531,Z 1185.454,A -85,B 0,C 180,E1 16739.998,E2 16739.998} C_VEL
LIN {X 0,Y 412.843,Z 1185.219,A -85,B 0,C 180,E1 16744.196,E2 16744.196} C_VEL
LIN {X 0,Y 413.905,Z 1180.554,A -85,B 0,C 180,E1 16749.226,E2 16749.226} C_VEL
LIN {X 0,Y 415.989,Z 1171.204,A -85,B 0,C 180,E1 16754.191,E2 16754.191} C_VEL
LIN {X 0,Y 420.17,Z 1155.59,A -85,B 0,C 180,E1 16759.428,E2 16759.428} C_VEL
LIN {X 0,Y 426.319,Z 1134.55,A -85,B 0,C 180,E1 16764.331,E2 16764.331} C_VEL
LIN {X 0,Y 434.483,Z 1107.737,A -85,B 0,C 180,E1 16768.85,E2 16768.85} C_VEL
LIN {X 0,Y 444.125,Z 1075.321,A -85,B 0,C 180,E1 16772.835,E2 16772.835} C_VEL
LIN {X 0,Y 454.936,Z 1037.096,A -85,B 0,C 180,E1 16776.272,E2 16776.272} C_VEL
LIN {X 0,Y 459.853,Z 1016.721,A -85,B 0,C 180,E1 16777.807,E2 16777.807} C_VEL
LIN {X 0,Y 459.61,Z 1001.962,A -85,B 0,C 180,E1 16779.854,E2 16779.854} C_VEL
LIN {X 0,Y 458.463,Z 992.395,A -85,B 0,C 180,E1 16782.21,E2 16782.21} C_VEL
LIN {X 0,Y 458.119,Z 989.674,A -85,B 0,C 180,E1 16783.84,E2 16783.84} C_VEL
LIN {X 0,Y 458.871,Z 991.703,A -85,B 0,C 180,E1 16786.422,E2 16786.422} C_VEL
LIN {X 0,Y 460.665,Z 999.632,A -85,B 0,C 180,E1 16788.607,E2 16788.607} C_VEL
LIN {X 0,Y 462.213,Z 1012.418,A -85,B 0,C 180,E1 16790.502,E2 16790.502} C_VEL
LIN {X 0,Y 460.199,Z 1022.629,A -85,B 0,C 180,E1 16791.124,E2 16791.124} C_VEL
LIN {X 0,Y 448.837,Z 1066.02,A -85,B 0,C 180,E1 16793.828,E2 16793.828} C_VEL
LIN {X 0,Y 438.62,Z 1104.249,A -85,B 0,C 180,E1 16797.164,E2 16797.164} C_VEL
LIN {X 0,Y 429.76,Z 1137.129,A -85,B 0,C 180,E1 16801.014,E2 16801.014} C_VEL
LIN {X 0,Y 422.537,Z 1165.653,A -85,B 0,C 180,E1 16805.476,E2 16805.476} C_VEL
LIN {X 0,Y 417.299,Z 1188.559,A -85,B 0,C 180,E1 16810.298,E2 16810.298} C_VEL
LIN {X 0,Y 414.288,Z 1205.504,A -85,B 0,C 180,E1 16815.228,E2 16815.228} C_VEL
LIN {X 0,Y 412.867,Z 1217.61,A -85,B 0,C 180,E1 16820.496,E2 16820.496} C_VEL
LIN {X 0,Y 412.575,Z 1224.105,A -85,B 0,C 180,E1 16825.818,E2 16825.818} C_VEL
LIN {X 0,Y 412.68,Z 1225.21,A -85,B 0,C 180,E1 16830.018,E2 16830.018} C_VEL
LIN {X 0,Y 412.66,Z 1222.651,A -85,B 0,C 180,E1 16834.218,E2 16834.218} C_VEL
LIN {X 0,Y 412.946,Z 1215.425,A -85,B 0,C 180,E1 16838.895,E2 16838.895} C_VEL
LIN {X 0,Y 413.963,Z 1201.055,A -85,B 0,C 180,E1 16844.282,E2 16844.282} C_VEL
LIN {X 0,Y 416.31,Z 1182.023,A -85,B 0,C 180,E1 16849.085,E2 16849.085} C_VEL
LIN {X 0,Y 419.617,Z 1160.78,A -85,B 0,C 180,E1 16853.065,E2 16853.065} C_VEL
LIN {X 0,Y 417.743,Z 1149.679,A -85,B 0,C 180,E1 16854.902,E2 16854.902} C_VEL
LIN {X 0,Y 415.814,Z 1137.737,A -85,B 0,C 180,E1 16856.659,E2 16856.659} C_VEL
LIN {X 0,Y 421.645,Z 1105.272,A -85,B 0,C 180,E1 16860.345,E2 16860.345} C_VEL
LIN {X 0,Y 427.896,Z 1067.218,A -85,B 0,C 180,E1 16863.508,E2 16863.508} C_VEL
LIN {X 0,Y 433.683,Z 1026.614,A -85,B 0,C 180,E1 16865.835,E2 16865.835} C_VEL
LIN {X 0,Y 434.907,Z 1009.306,A -85,B 0,C 180,E1 16866.622,E2 16866.622} C_VEL
LIN {X 0,Y 419.655,Z 966.8,A -85,B 0,C 180,E1 16869.171,E2 16869.171} C_VEL
LIN {X 0,Y 402.396,Z 923.03,A -85,B 0,C 180,E1 16871.821,E2 16871.821} C_VEL
LIN {X 0,Y 402.32,Z 923.03,A -85,B 0,C 180,E1 16878.716,E2 16878.716} C_VEL
LIN {X 0,Y 402.486,Z 923.03,A -85,B 0,C 180,E1 16885.728,E2 16885.728} C_VEL
LIN {X 0,Y 402.624,Z 923.03,A -85,B 0,C 180,E1 16890.8,E2 16890.8} C_VEL
LIN {X 0,Y 402.904,Z 923.03,A -85,B 0,C 180,E1 16897.975,E2 16897.975} C_VEL
LIN {X 0,Y 403.066,Z 923.03,A -85,B 0,C 180,E1 16902.197,E2 16902.197} C_VEL
LIN {X 0,Y 405.581,Z 928.746,A -85,B 0,C 180,E1 16902.777,E2 16902.777} C_VEL
LIN {X 0,Y 419.196,Z 957.347,A -85,B 0,C 180,E1 16905.423,E2 16905.423} C_VEL
LIN {X 0,Y 425.616,Z 977.355,A -85,B 0,C 180,E1 16906.698,E2 16906.698} C_VEL
LIN {X 0,Y 424.269,Z 1015.495,A -85,B 0,C 180,E1 16907.924,E2 16907.924} C_VEL
LIN {X 0,Y 421.9,Z 1044.778,A -85,B 0,C 180,E1 16909.686,E2 16909.686} C_VEL
LIN {X 0,Y 418.677,Z 1069.961,A -85,B 0,C 180,E1 16912.093,E2 16912.093} C_VEL
LIN {X 0,Y 415.288,Z 1090.365,A -85,B 0,C 180,E1 16915.045,E2 16915.045} C_VEL
LIN {X 0,Y 412.068,Z 1105.803,A -85,B 0,C 180,E1 16918.426,E2 16918.426} C_VEL
LIN {X 0,Y 409.37,Z 1115.912,A -85,B 0,C 180,E1 16922.118,E2 16922.118} C_VEL
LIN {X 0,Y 408.321,Z 1119.156,A -85,B 0,C 180,E1 16924.247,E2 16924.247} C_VEL
LIN {X 0,Y 407.445,Z 1120.706,A -85,B 0,C 180,E1 16926.39,E2 16926.39} C_VEL
LIN {X 0,Y 406.928,Z 1120.548,A -85,B 0,C 180,E1 16928.544,E2 16928.544} C_VEL
LIN {X 0,Y 406.723,Z 1116.125,A -85,B 0,C 180,E1 16932.337,E2 16932.337} C_VEL
LIN {X 0,Y 407.082,Z 1106.308,A -85,B 0,C 180,E1 16936.167,E2 16936.167} C_VEL
LIN {X 0,Y 408.012,Z 1090.819,A -85,B 0,C 180,E1 16939.754,E2 16939.754} C_VEL
LIN {X 0,Y 409.438,Z 1070.355,A -85,B 0,C 180,E1 16942.92,E2 16942.92} C_VEL
LIN {X 0,Y 410.933,Z 1045.153,A -85,B 0,C 180,E1 16945.554,E2 16945.554} C_VEL
LIN {X 0,Y 412.377,Z 1016.82,A -85,B 0,C 180,E1 16947.485,E2 16947.485} C_VEL
LIN {X 0,Y 413.116,Z 986.223,A -85,B 0,C 180,E1 16948.671,E2 16948.671} C_VEL
LIN {X 0,Y 412.266,Z 966.627,A -85,B 0,C 180,E1 16949.149,E2 16949.149} C_VEL
LIN {X 0,Y 402.851,Z 923.03,A -85,B 0,C 180,E1 16950.541,E2 16950.541} C_VEL
LIN {X 0,Y 402.304,Z 923.03,A -85,B 0,C 180,E1 16957.904,E2 16957.904} C_VEL
LIN {X 0,Y 402.332,Z 923.03,A -85,B 0,C 180,E1 16964.449,E2 16964.449} C_VEL
LIN {X 0,Y 402.34,Z 923.03,A -85,B 0,C 180,E1 16970.301,E2 16970.301} C_VEL
LIN {X 0,Y 402.459,Z 923.03,A -85,B 0,C 180,E1 16975.703,E2 16975.703} C_VEL
LIN {X 0,Y 402.827,Z 923.03,A -85,B 0,C 180,E1 16983.228,E2 16983.228} C_VEL
LIN {X 0,Y 403.115,Z 923.03,A -85,B 0,C 180,E1 16990.265,E2 16990.265} C_VEL
LIN {X 0,Y 403.483,Z 923.03,A -85,B 0,C 180,E1 16996.996,E2 16996.996} C_VEL
LIN {X 0,Y 403.954,Z 923.03,A -85,B 0,C 180,E1 17003.538,E2 17003.538} C_VEL
LIN {X 0,Y 404.483,Z 923.03,A -85,B 0,C 180,E1 17009.981,E2 17009.981} C_VEL
LIN {X 0,Y 403.991,Z 923.03,A -85,B 0,C 180,E1 17016.423,E2 17016.423} C_VEL
LIN {X 0,Y 403.519,Z 923.03,A -85,B 0,C 180,E1 17023.173,E2 17023.173} C_VEL
LIN {X 0,Y 403.137,Z 923.03,A -85,B 0,C 180,E1 17029.694,E2 17029.694} C_VEL
LIN {X 0,Y 402.82,Z 923.03,A -85,B 0,C 180,E1 17036.73,E2 17036.73} C_VEL
LIN {X 0,Y 402.6,Z 923.03,A -85,B 0,C 180,E1 17041.674,E2 17041.674} C_VEL
LIN {X 0,Y 402.368,Z 923.03,A -85,B 0,C 180,E1 17047.936,E2 17047.936} C_VEL
LIN {X 0,Y 402.402,Z 923.03,A -85,B 0,C 180,E1 17054.477,E2 17054.477} C_VEL
LIN {X 0,Y 402.507,Z 923.03,A -85,B 0,C 180,E1 17059.323,E2 17059.323} C_VEL
LIN {X 0,Y 419.259,Z 969.271,A -85,B 0,C 180,E1 17062.285,E2 17062.285} C_VEL
LIN {X 0,Y 430.942,Z 1007.731,A -85,B 0,C 180,E1 17065.227,E2 17065.227} C_VEL
LIN {X 0,Y 430.885,Z 1017.074,A -85,B 0,C 180,E1 17065.865,E2 17065.865} C_VEL
LIN {X 0,Y 425.015,Z 1055.232,A -85,B 0,C 180,E1 17068.762,E2 17068.762} C_VEL
LIN {X 0,Y 419.291,Z 1088.359,A -85,B 0,C 180,E1 17072.206,E2 17072.206} C_VEL
LIN {X 0,Y 413.952,Z 1117.859,A -85,B 0,C 180,E1 17076.323,E2 17076.323} C_VEL
LIN {X 0,Y 409.586,Z 1143.347,A -85,B 0,C 180,E1 17081.164,E2 17081.164} C_VEL
LIN {X 0,Y 406.788,Z 1161.813,A -85,B 0,C 180,E1 17086.025,E2 17086.025} C_VEL
LIN {X 0,Y 405.414,Z 1174.729,A -85,B 0,C 180,E1 17090.92,E2 17090.92} C_VEL
LIN {X 0,Y 404.776,Z 1182.543,A -85,B 0,C 180,E1 17095.716,E2 17095.716} C_VEL
LIN {X 0,Y 404.66,Z 1185.845,A -85,B 0,C 180,E1 17099.998,E2 17099.998} C_VEL
LIN {X 0,Y 404.969,Z 1185.745,A -85,B 0,C 180,E1 17104.278,E2 17104.278} C_VEL
LIN {X 0,Y 406.272,Z 1180.64,A -85,B 0,C 180,E1 17109.871,E2 17109.871} C_VEL
LIN {X 0,Y 408.939,Z 1169.89,A -85,B 0,C 180,E1 17115.411,E2 17115.411} C_VEL
LIN {X 0,Y 413.898,Z 1153.081,A -85,B 0,C 180,E1 17120.85,E2 17120.85} C_VEL
LIN {X 0,Y 421.116,Z 1130.468,A -85,B 0,C 180,E1 17125.891,E2 17125.891} C_VEL
LIN {X 0,Y 429.848,Z 1103.704,A -85,B 0,C 180,E1 17130.239,E2 17130.239} C_VEL
LIN {X 0,Y 440.511,Z 1070.664,A -85,B 0,C 180,E1 17134.195,E2 17134.195} C_VEL
LIN {X 0,Y 451.818,Z 1033.373,A -85,B 0,C 180,E1 17137.449,E2 17137.449} C_VEL
